// TwinCAT 3 PLC project HPT_PLC
// Title: Hardpoint Test Stand
// Company: GTMO
// Author: A. Everman, T. Ranka
// ProjectVersion: 1.4.5
// ProgramVersion: 3.1.4024.12
// libraries:
//   CmpBitmapPool, * (System)
//   Tc2_ControllerToolbox, * (Beckhoff Automation GmbH)
//   Tc2_EtherCAT, * (Beckhoff Automation GmbH)
//   Tc2_SerialCom, * (Beckhoff Automation GmbH)
//   Tc2_Standard, * (Beckhoff Automation GmbH)
//   Tc2_System, * (Beckhoff Automation GmbH)
//   Tc2_Utilities, * (Beckhoff Automation GmbH)
//   Tc3_Module, * (Beckhoff Automation GmbH)
// project tree:
//   DUTs/ ImagePool.TcIPO (not stored)
//   / Fast.TcTTO, GlobalTextList.TcGTLO, PlcTask.TcTTO, Visualization Manager.TcVMO (not stored)
//   GVLs/ GVL_TS.TcGVL
//   POUs/ FB_AirConv.TcPOU, Background.TcPOU, BackgroundEL.TcPOU, FB_BinToVer.TcPOU, FB_ClearFault.TcPOU, FB_CountConv.TcPOU, FB_PLCTime.TcPOU, FB_PyListener.TcPOU, FB_PyListenerStiffness.TcPOU, FB_PyPosRep.TcPOU, FB_ReadAlias.TcPOU, FB_ReadNcyl.TcPOU, FB_ReadSig.TcPOU, FB_readtextfile.TcPOU, FB_SAstiffness.TcPOU, FB_SaveData.TcPOU, FB_SerialCom.TcPOU, FB_HeidConv.TcPOU, FB_TriForce.TcPOU, FB_WriteHPTSettings.TcPOU, FB_WritePWM.TcPOU, FB_WriteSDO.TcPOU, MAIN.TcPOU, FB_MtrCtrl.TcPOU, FB_PLoop.TcPOU, FB_ROMTest.TcPOU, FB_SineSweep.TcPOU
// real-time tasks:
//   TASK PlcTask: cycle T#1ms, priority 6, ADS port 350
//   TASK Fast: cycle T#1ms, priority 4, ADS port 351
// motion (NC):
//   TASK NC-Task 1 SAF: cycle T#2ms, priority 8, ADS port 501
//   TASK NC-Task 1 SVB: cycle T#10ms, priority 12, ADS port 511
//   AXIS Axis 1 (id 1)
//     OtherSettings: AllowMotionCmdToSlave=true
//     encoder EncType=19
//       EncPara: MaxCount=#xffffffff
//     drive DrvType=16
//       DrvPara: MaxCount=#xffffffff
//         Analog: TorqueSetpointScale=10, ScaleFactorActTorque=0.1
//         TimeComp: TaskDelayCycles=1
//     controller CtrType=1
//       CtrPara: PriorControlFactor=1
//         Observer: BandWidth=20
// I/O:
//   DEVICE Device 1 (EtherCAT), AmsNetId 10.10.160.129.2.1
//     Term 2 (EK1100) [EK1100 EtherCAT Coupler (2A E-Bus)]
//       Term 13 (EL6070-0033) [EL6070-0033 1Ch. Licence key terminal, individual licences]
//       Term 14 (EL4102) [EL4102 2Ch. Ana. Output  0-10V, 16bit]
//       Term 16 (EL3002) [EL3002 2Ch. Ana. Input +/-10V]
//       Term 18 (EL3052) [EL3052 2Ch. Ana. Input 4-20mA]
//       Term 19 (EL5101) [EL5101 1Ch. Inc. Encoder 5V]
//       Term 29 (EL9011) [EL9011 End Terminal]
//     Drive 20 (BEL) [BEL]
//       modules: Module 1 (Cyclic velocity Mode)
//     Term 21 (EK1100) [EK1100 EtherCAT Coupler (2A E-Bus)]
//       Term 22 (EL5042) [EL5042 2Ch. BiSS-C Encoder]
//       Term 23 (EL3312) [EL3312 2Ch. Ana. Input Thermocouple (TC)]
//       Term 24 (EL9505) [EL9505 Power supply terminal 5V]
//       Term 26 (EL3356-0010) [EL3356-0010 1Ch. Ana. Input Resistor Bridge Terminal, 24bit, High Precision]
//       Term 30 (EL9011) [EL9011 End Terminal]
//     Box 17 (m1sa) [m1sa]
// variable links:
//   HPT_PLC/HPT_PLC Instance <-> Device 1 (EtherCAT)/Box 17 (m1sa)
//     PlcTask Inputs/MAIN.err_cal <-> Status process data mapping/MAIN.err_cal
//     PlcTask Inputs/MAIN.err_dongle <-> Status process data mapping/MAIN.err_dongle
//     PlcTask Inputs/MAIN.err_f_minmax <-> Status process data mapping/MAIN.err_f_minmax
//     PlcTask Inputs/MAIN.err_f_step <-> Status process data mapping/MAIN.err_f_step
//     PlcTask Inputs/MAIN.err_locid <-> Status process data mapping/MAIN.err_locid
//     PlcTask Inputs/MAIN.err_mhb <-> Status process data mapping/MAIN.err_mhb
//     PlcTask Inputs/MAIN.err_soc <-> Status process data mapping/MAIN.err_soc
//     PlcTask Inputs/MAIN.pwm1 <-> Status process data mapping/MAIN.pwm1
//     PlcTask Inputs/MAIN.rb_x <-> Status process data mapping/MAIN.rb_x
//     PlcTask Inputs/MAIN.spr_x <-> Status process data mapping/MAIN.spr_x
//     PlcTask Outputs/MAIN.close_loop <-> Control process data mapping/MAIN.close_loop
//     PlcTask Outputs/MAIN.enable <-> Control process data mapping/MAIN.enable
//     PlcTask Outputs/MAIN.msthb <-> Control process data mapping/MAIN.msthb
//     PlcTask Outputs/MAIN.sp_x <-> Control process data mapping/MAIN.sp_x
//   HPT_PLC/HPT_PLC Instance <-> Device 1 (EtherCAT)/Drive 20 (BEL)
//     PlcTask Inputs/GVL_TS.DIO_status <-> Transmit PDO 4/GVL_TS.DIO_status
//     PlcTask Inputs/GVL_TS.EncoderFault <-> Transmit PDO 3/GVL_TS.EncoderFault
//     PlcTask Inputs/GVL_TS.Sticky <-> Transmit PDO 4/GVL_TS.Sticky
//     PlcTask Inputs/GVL_TS.cmdVel <-> Transmit PDO 1/GVL_TS.cmdVel
//     PlcTask Inputs/GVL_TS.mtrCurrent <-> Transmit PDO 3/GVL_TS.mtrCurrent
//     PlcTask Inputs/GVL_TS.mtr_pos <-> Transmit PDO 2/GVL_TS.mtr_pos
//     PlcTask Inputs/GVL_TS.mtr_tor <-> Module 1 (Cyclic velocity Mode)/Cyclic velocity Inputs/GVL_TS.mtr_tor
//     PlcTask Inputs/GVL_TS.mtrl_vel <-> Module 1 (Cyclic velocity Mode)/Cyclic velocity Inputs/GVL_TS.mtrl_vel
//     PlcTask Inputs/GVL_TS.status_word <-> Module 1 (Cyclic velocity Mode)/Cyclic velocity Inputs/GVL_TS.status_word
//     PlcTask Outputs/GVL_TS.ClearLatched2181 <-> Receive PDO 4/GVL_TS.ClearLatched2181
//     PlcTask Outputs/GVL_TS.ClearLatched2183 <-> Receive PDO 4/GVL_TS.ClearLatched2183
//     PlcTask Outputs/GVL_TS.StopAbort <-> Receive PDO 3/GVL_TS.StopAbort
//     PlcTask Outputs/GVL_TS.TransitionFromQS <-> Receive PDO 3/GVL_TS.TransitionFromQS
//     PlcTask Outputs/GVL_TS.control_word <-> Module 1 (Cyclic velocity Mode)/Cyclic velocity Outputs/GVL_TS.control_word
//     PlcTask Outputs/GVL_TS.target_vel <-> Module 1 (Cyclic velocity Mode)/Cyclic velocity Outputs/GVL_TS.target_vel
//     PlcTask Outputs/MAIN.FaultMask <-> Receive PDO 3/MAIN.FaultMask
//   HPT_PLC/HPT_PLC Instance <-> Device 1 (EtherCAT)/Term 2 (EK1100)/Term 14 (EL4102)
//     PlcTask Outputs/GVL_TS.AirOut1 <-> Channel 1/GVL_TS.AirOut1
//     PlcTask Outputs/GVL_TS.AirOut2 <-> Channel 2/GVL_TS.AirOut2
//   HPT_PLC/HPT_PLC Instance <-> Device 1 (EtherCAT)/Term 2 (EK1100)/Term 16 (EL3002)
//     PlcTask Inputs/GVL_TS.LazrStrength <-> AI Standard Channel 1/GVL_TS.LazrStrength
//   HPT_PLC/HPT_PLC Instance <-> Device 1 (EtherCAT)/Term 2 (EK1100)/Term 18 (EL3052)
//     PlcTask Inputs/GVL_TS.FlowIn <-> AI Standard Channel 2/GVL_TS.FlowIn
//     PlcTask Inputs/GVL_TS.PressureIn <-> AI Standard Channel 1/GVL_TS.PressureIn
//   HPT_PLC/HPT_PLC Instance <-> Device 1 (EtherCAT)/Term 21 (EK1100)/Term 22 (EL5042)
//     PlcTask Inputs/GVL_TS.ActEncCount <-> FB Inputs Channel 1/GVL_TS.ActEncCount
//     PlcTask Inputs/GVL_TS.MirEncCount <-> FB Inputs Channel 2/GVL_TS.MirEncCount
//   HPT_PLC/HPT_PLC Instance <-> Device 1 (EtherCAT)/Term 21 (EK1100)/Term 23 (EL3312)
//     PlcTask Inputs/GVL_TS.EncTapeTemp <-> TC Inputs Channel 1/GVL_TS.EncTapeTemp
//     PlcTask Inputs/GVL_TS.MotorTemp <-> TC Inputs Channel 2/GVL_TS.MotorTemp
//   HPT_PLC/HPT_PLC Instance <-> Device 1 (EtherCAT)/Term 21 (EK1100)/Term 26 (EL3356-0010)
//     PlcTask Inputs/GVL_TS.LC_InR <-> RMB Value (Real)/GVL_TS.LC_InR

CONFIGURATION HPT_PLC
    RESOURCE PLC ON TwinCAT3
        TASK Fast(INTERVAL := T#1ms, PRIORITY := 4);
        TASK PlcTask(INTERVAL := T#1ms, PRIORITY := 6);
        PROGRAM Background WITH Fast : Background;
        PROGRAM MAIN WITH PlcTask : MAIN;
    END_RESOURCE
END_CONFIGURATION

// ---- GVLs/GVL_TS.TcGVL
VAR_GLOBAL CONSTANT
	max_rows : UDINT := 10001;
END_VAR

{attribute 'qualified_only'}
VAR_GLOBAL

// Variables for EL4102 0-10V Module for Air Control
AirOut1 AT %Q*			: INT;
AirOut2 AT %Q*			: INT;

// Variables for EL5101 RS422 Incremental Encoder Interface
RSCount AT %I* 			: DINT;
CountReset AT %Q* 		: DINT; // Count reset variable, set to zero for tareing of laser interferometer 
CountResetEn AT %Q* 	: BOOL; // Enable flag for counter reset
LaserUnder AT %I* 		: BOOL; // Underflow flag for debugging
LaserOver AT %I* 		: BOOL; // Overflow flag for debugging

// Variables for HPT eBox EL5042 BiSS-C Encoder Interface
ActEncCount AT %I* 		: ULINT;
MirEncCount AT %I* 		: ULINT;

// Motor variables
mtr_tor AT %I* 			: INT;
StopAbort AT %Q* 		: INT;
TransitionFromQS AT %Q* : INT;
mtrCurrent AT %I* 		: INT;
control_word AT %Q* 	: UINT;
status_word AT %I* 		: UINT;
target_vel AT %Q* 		: DINT :=0; (*0.1cnts/s*)
mtrl_vel AT %I* 		: DINT; (*0.1cnts/sec*)
mtr_pos AT %I* 			: DINT; (*counts*)
velLoopErr AT %I*		: DINT;
cmdVel AT %I*			: DINT;
ClearLatched2181 AT %Q* : UDINT;
ClearLatched2183 AT %Q* : UDINT;
Sticky AT %I* 			: UDINT;
EncoderFault AT %I* 	: UDINT;
DIO_status AT %I* 		: UDINT;	(*limit switch status*)
bLim_pos 				: BOOL := FALSE;
bLim_neg 				: BOOL := FALSE;
bEnableState 			: BOOL;
bReset 					: BOOL;
bEnable 				: BOOL;
sJog 					: STRING;

// Load cell input variable
LC_InR AT %I* 			: REAL;
LC_Tara AT %Q*			: BYTE;

// Thermocouple Variables
EncTapeTemp AT %I* 		: INT;
MotorTemp AT %I* 		: INT;

// Limit switch triggered status variables
bPos 					: BOOL;
bNeg 					: BOOL;
Pdiff 					: LREAL;

// EL3002 Interferometer Laser Strength Indicator Variable
LazrStrength AT %I* 	: INT;

// EL3052 4...20mA analog input variables for pressure/flow sensors
PressureIn AT %I* 		: INT;
FlowIn AT %I* 			: INT;

// Buffer variable for RS-232 COM port
RxBufferEL				: ComBuffer;	(* Receive data buffer; used with all receive function blocks *)
TxBufferEL				: ComBuffer;	(* Transmit data buffer; used with all receive function blocks *)

(* DEBUG VARIABLES *)
//bTEST1 				: BOOL := FALSE;
//bTEST2 				: BOOL := FALSE;
//wTest 				: WORD;
//sTest 				: STRING;

END_VAR

// ---- POUs/Background.TcPOU
PROGRAM Background
VAR
END_VAR

(*
The SerialLineControl function block is supposed to be called in every PLC cycle.
It communicates with the serial line hardware device and transmits or receives data.
The SerialLineControl can be called in the standard task (e.g.for PcCOM port usage) 
or in a separate fast task (e.g.for terminal usage) as well.
A fast separate task will be necessary at high baud rates or with KL6001 terminals 
which have a small process image (3 or 5 data bytes only)
*)

(* background communication with the EL6001 terminal *)
BackgroundEL();

END_PROGRAM

// ---- POUs/BackgroundEL.TcPOU
PROGRAM BackgroundEL
VAR
	(* background communication with the EL6001 terminal *)
	fbEL6001Ctrl		: SerialLineControl;
	bEL6001CtrlError	: BOOL;
	eEL6001CtrlErrorID	: ComError_t;
	(* 	I/O variables for a EL6001 terminal*)
	stIn_EL6001 AT %I*	: EL6inData22B;	(* linked to the EL6001 in the TwinCAT System Manager *)
	stOut_EL6001 AT %Q*	: EL6outData22B;(* linked to the EL6001 in the TwinCAT System Manager *)
END_VAR

(*
The SerialLineControl function block is supposed to be called in every PLC cycle.
It communicates with the serial line hardware device and transmits or receives data.
The SerialLineControl can be called in the standard task (e.g.for PcCOM port usage) 
or in a separate fast task (e.g.for terminal usage) as well.
A fast separate task will be necessary at high baud rates or with KL6001 terminals 
which have a small process image (3 or 5 data bytes only)
*)

(* background communication with the EL6001 terminal *)
fbEL6001Ctrl(
	Mode:= SERIALLINEMODE_EL6_22B, 
	pComIn:= ADR(stIn_EL6001), 
	pComOut:= ADR(stOut_EL6001), 
	SizeComIn:= SIZEOF(stIn_EL6001), 
	Error=> , 
	ErrorID=> , 
	TxBuffer:= GVL_TS.TxBufferEL, 
	RxBuffer:= GVL_TS.RxBufferEL );
IF fbEL6001Ctrl.Error THEN
	bEL6001CtrlError := TRUE;
	eEL6001CtrlErrorID := fbEL6001Ctrl.ErrorID;
END_IF

END_PROGRAM

// ---- POUs/MAIN.TcPOU
PROGRAM MAIN
VAR

// Function instants
	fbSAstiffness		: FB_SAstiffness;
	fbWriteSettings		: FB_WriteHPTSettings;
	fbROM 				: FB_ROMTest;
	fbSWEEP 			: FB_SineSweep;
	fbSTIFF 			: FB_TriForce;
	fbBWY				: FB_TriForce;
	fbPLOOP 			: FB_PLoop;
	fbToString 			: FB_FormatString;
	fbB2V 				: FB_BinToVer;
	fbEL6001 			: FB_SerialCom;
	fbHeidCon 			: FB_HeidConv;
	fbPyListen			: FB_PyListener;
	fbPyListenStiff		: FB_PyListenerStiffness;
	fbWriteSDO			: FB_WriteSDO;
	fbGetTime			: FB_PLCTime;
	fbPyPosRep			: FB_PyPosRep;
	
// Startup Variables
	FaultMask AT %Q* 	: UDINT := 2#00000000;
	
// HMI Variables
	txtLazer 			: STRING;
	txtActEncVal 		: STRING;
	txtMirEncVal 		: STRING;
	txtRPM 				: STRING;
	txtTorque 			: STRING;
	BinStatus 			: STRING;
	txtActROM 			: STRING;
	txtMirROM 			: STRING;
	txtEngActEnc 		: STRING; 
	txtEngMirEnc 		: STRING;
	txtActMid 			: STRING;
	txtMirMid 			: STRING;
	txtLC 				: STRING;
	txtPdiff 			: STRING;
	txtBWYPress 		: STRING;
	txtFlow 			: STRING;
	txtMtrTemp			: STRING;
	txtEncTemp			: STRING;
	txtMtrCurrent		: STRING;
	sHeidOut 			: STRING;
	HeidA 				: STRING;
	HeidB 				: STRING;
	HeidC 				: STRING;
	HeidD 				: STRING;
	sSetpoint 			: STRING;
	sSelHPT				: STRING;
	sTime				: STRING;
	sp_force 			: STRING;
	engActEnc 			: LREAL; // Converted engineering units
	engMirEnc 			: LREAL; // Converted engineering units
	mtrRPM 				: LREAL;
	BWYPressPSI			: REAL;
	FlowRate 			: REAL;
	mtrTorq 			: REAL;
	mtrCurrent			: REAL;
	LazrMeter 			: REAL;
	AIR_CTR 			: REAL;
	ROM_Act 			: REAL;
	ROM_mirr			: REAL;
	HeidANum 			: REAL;
	HeidBNum 			: REAL;
	HeidCNum 			: REAL;
	HeidDNum 			: REAL;
	COARSE_VAL 			: REAL; // Variables for converted interferometer converted counts to length
	FINE_VAL 			: REAL;
	MtrTemp				: REAL;
	EncTemp				: REAL;
	TestCycles			: INT;
	atto1 				: REAL;
	atto2 				: REAL;
	atto3 				: REAL;
	atto4 				: REAL;
	atto5 				: REAL;
	atto6 				: REAL;
	atto1uM 			: REAL;
	atto2uM 			: REAL;
	atto3uM 			: REAL;
	atto4uM 			: REAL;
	atto5uM 			: REAL;
	atto6uM 			: REAL;
	satto1uM 			: STRING;
	satto2uM 			: STRING;
	satto3uM 			: STRING;
	satto4uM 			: STRING;
	satto5uM 			: STRING;
	satto6uM 			: STRING;
	ROM_ActMid 			: ULINT;
	ROM_MirrMid 		: ULINT;
	btnEnb 				: BOOL;
	btnEnbnum 			: BOOL := FALSE;
	btnReset 			: BOOL := FALSE;
	btnTareLC			: BOOL := FALSE;
	btnPyPosRep			: BOOL := FALSE;
	btnClrSAerrors		: BOOL := FALSE; 
	tglSine 			: BOOL := FALSE;
	tglROM 				: BOOL := FALSE;
	tglStiffness 		: BOOL := FALSE;
	tglSAstiffness		: BOOL := FALSE;
	tglBWY				: BOOL := FALSE;
	tglPLoop 			: BOOL := FALSE;
	tglPyTest			: BOOL := FALSE;
	JogPos 				: BOOL := FALSE;
	JogNeg 				: BOOL := FALSE;
	PyLoad				: BOOL;
	PyLoadBusy			: BOOL := FALSE;
	PyEnable			: BOOL := TRUE;
	MtrErrArr 			: ARRAY[0..15] OF BOOL;
	
(* DEBUG VARIABLES *)
	//test 				: BOOL := FALSE;
	//int1 				: INT;
	//real2 			: REAL;
	//real3 			: REAL;
	
// SA Related Variables for Stiffness Fixture
	// actions
	actions : (idle, clear_all, enable_all, disable_all,read_ncyl,read_alias,read_gains,write_gains,read_file,send_waveform_cmd, send_waveform_cmd_debug, send_waveform_pwm);
	sp_x AT %Q* : REAL;
	sp_y AT %Q* : REAL;
	sp_z AT %Q* : REAL;
	
	f_num : INT := 1; // file number
	signal_scale : REAL := 1;
	signal_offset : REAL :=0;
	signal_axis : INT :=1;

	//VARIABLES FOR SENSOR OUTPUTS TO BE DISPLAYED IN UNITS OF MEASUREMENT
	spr_x AT %I* : REAL;
	spr_y AT %I* : REAL;
	spr_z AT %I* : REAL;
	rb_x AT %I* : REAL;
	txtRB_X 	: STRING;
	rb_y AT %I* : REAL;
	rb_z AT %I* : REAL;
	pwm1 AT %I* : REAL;
	pwm2 AT %I* : REAL;
	pwm3 AT %I* : REAL;
	cyl_sum : REAL;
	cmd_sum : REAL;
	
	//CONSTANTS FOR ADC GAIN COEFFICIENTS
	//ADC1: CH1 and CH2 PRESSURE, CH3 FLOW, CH4 NOT CONNECTED
	//ADC2: ALL CHANNELS PRESSURE
	GAIN_PRESSURE : REAL := 2.2;
	GAIN_FLOW : REAL := 2.2;//80;
	
	// ***********************************************************
	
	sa_addr : UINT := 1013;	
	clearfault : FB_ClearFault;
	readncyl : FB_ReadNcyl;
	readalias : FB_ReadAlias;
	readfile : FB_readtextfile;
	
	max_rows : UDINT := 10001;
	sfile : T_MaxString ;
	waveform_pwm : FB_WritePWM;
	state : INT := 2;
	step : DWORD :=0;
	bError : BOOL;
	t_index : UINT :=1;
	alias : UDINT;
	ncyl: UINT;
	signal : ARRAY[1.. GVL_TS.max_rows] OF REAL;
	
	fol_err : REAL;
	db : REAL := 14.0;
	dbi : REAL := 0;
	pwm : REAL := 0.0;
	value : REAL := 0.0;
	
	sdo_address: UINT;
	subIndex: BYTE;
	sNetId_local : T_AmsNetId := '10.134.198.192.2.1';	// Address of this computer 
	//sNetId_local : T_AmsNetId := '10.10.16.19.2.1';	// Address of this computer
	
// heartbeat
	msthb AT %Q* : UDINT;
	enable AT %Q* : BOOL;
	close_loop AT %Q* : BOOL;
	
	err_mhb AT %I* : BOOL;
	err_f_minmax AT %I* : BOOL;
	err_f_step AT %I* : BOOL;
	err_cal AT %I* : BOOL;
	err_dongle AT %I* : BOOL;
	err_locid AT %I* : BOOL;
	err_soc AT %I* : BOOL;
	err_ff AT %I* : BOOL;
	
	force : INT;

END_VAR

(*-----------------------------------------------------------------------------------------------------
 	Hardpoint Test Stand, GMTO
 	v2.2.0
	
	*CHANGE LOG*
	1.0.0
			- First "complete" release
				-HMI
					-Control and monitor all sensors and tests
				-Scope project
					-Monitor and record all availible sensors and ADS variables and export as CSV for analysis
				-Tests included:
					-Range of motion
					-Position loop
					-Stiffness test
						-Multiple force profiles availible
					-Sine sweep
						*NOT TESTED ON HARDWARE, WORKS IN SCOPE PROJECT ONLY*
					
	1.4.5: 
			- Refactoring started:
				Clean up variables by standardizing naming conventions (upper camel case, leading lowercase b, s, fb, etc. for special case variables) 
				Whitespaces in declarations
				Removing unused variables
				Change variable types to lower memory footprint
				Reorganize variables to group by type
				
	1.4.6
			- Thermocouple data added to HMI
				Settings made in EL3312 to read correctly:
					CoE 8000:01 = TRUE
						8000:07 = TRUE
						8000:08 = TRUE
						8000:12 = 31451
						8000:13 = -730
						8000:14 = 4820
						8010:01 = TRUE
						8010:07 = TRUE
						8010:08 = TRUE
						8010:12 = 31438
						8010:13 = -730
						8010:14 = 4820
			- Further refactoring
			- Divided MAIN into clearer sections for ease of reading
			- Removed redundant limit switch check
			- Changed some HMI readouts to 4 decimal places
			
	1.4.7
			- HMI Cleanup and fixes
			- NOTE ADDED: EL5042 changes to be made to enable correct operation
				CoE 8008:15 - 26
					8008:16 - 0
					8018:15 - 26
					8018:16 - 0
	
	1.4.8	
			-= VERSION SKIPPED =-
	
	1.4.9	
			- Added, then removed, auto-tare for interferometer and load cell on test starts 
			- Added Tare button to HMI; disabled for time being
	
	2.0.0	
			- Python "PyListener" code added to listen for TC3 variables over ADS and build .CSV
				- Also grabs AttoCube measurements to calculate stiffness
			- Added ability to tare load cell back into HMI
				- Uses new FB_WriteSDO POU to write to SDOs in order to accomplish this
			- Added seperate buttons for both stiffness and breakaway tests
			- Simplified underlying stiffness/breakaway test code into one, singular function
				- Able to define both slope and force as inputs to function
			- Partitioned off tests into distinct "types" on HMI
			- Removed "Sine Sweep" test button from HMI; did not remove underlying code
				- CME has the ability to run bandwith tests natively, will need to add back into stand eventually
			- Further refactoring done to clean up unused variables/functions
			
	2.1.0
			- Python "PyListener" launches on start of any test, and ends collection on test stop
			- Further refactoring
			- Converted PLC time code into POU to clean up MAIN
	2.2.0
			- Added ability to toggle PyListener on and off
				- Buttons added on HMI for this
			- Able to launch PyListener for arbitrary data collection
			- Added cycle counter for stiffness/breakaway tests and readout on HMI
			- HMI cleaned up for better readability
			- HMI size property fixed to always show full dashboard when undocked
				
				
	TO-DO:
			
			- Use new FB_WriteSDO to force write all required settings on startup
				- Needs ability to write different variable sizes/types to correct positions
			- Continue refactoring as needed
			- Write new POU force stiffness/breakaway tests that has a "ramp up/hold/ramp down/hold/repeat profile"
				with ability to fully customize ramp speeds, hold times, and total force applied during all phases of test run
			- Possibly write a fully automated, non-steady state position loop test (I.E. start at set point, move up XXXcts, 
				return to starting setpoint, move down XXXcts, return to setpoint; do for how ever many cycles, each cycle
				being YYY[s] long)
			- Test/Debug Sine Sweep test on actual hardware
			- ??? (add to as necessary)

(*-----------------------------------------------------------------------------------------------------*)
 	Austin Everman - Overall framework, HMI, integration of code for individual tests, PyListener (with
	Trupti Ranka - coding for individual tests, technical help
	William Schoenell - AttoCube Python connection code

              _______________
          ==c(___(o(______(_()
                  \=\
                   )=\
                  //|\\
                 //|| \\
                // ||  \\
               //  ||   \\
              //         \\
			  
-------------------------------------------------------------------------------------------------------*)
(*-----------------------------------------------------------------------------------------------------*)
//fbWriteSettings();
(*-----------------------------------------------------------------------------------------------------*)
(* CONVERSION SECTION OF THE HMI THAT DEALS WITH TAKING RAW DATA AND CONVERTING IT FOR *)
(* DISPLAY ON THE DASHBOARD 														   *)
(*-----------------------------------------------------------------------------------------------------*)
// Parse status word into boolean array for HMI
fbB2V(
	BinInput := GVL_TS.status_word, 
	MtrErrArr => MtrErrArr
);
(*-----------------------------------------------------------------------------------------------------*)
// Convert interferometer signal strength voltage output to scaled 0-100% output for HMI
LazrMeter := (INT_TO_REAL(GVL_TS.LazrStrength)/32767) * 1000;
(*-----------------------------------------------------------------------------------------------------*)
// Call function to convert interferometer counts to mm
FB_CountConv(
	GVL_TS.RsCount, 
	MEASC_OUT => COARSE_VAL, // Return from function for conversion for coarse resolution laser intererometric measurements; Currently in use
	MEASF_OUT => FINE_VAL    // Not in use, but conversion made for fine resolution in event of use; setting is made on RLU dip switch on front of unit
);
(*-----------------------------------------------------------------------------------------------------*)
// Convert coarse interferometer value to string, limit to 6 decimal places for HMI, include 'traveling' engineering unit
fbToString(
	sFormat := '%.6f', 
	arg1 := F_REAL(COARSE_VAL), 
	sOut => txtLazer
);
txtLazer := CONCAT(txtLazer, ' mm');
(*-----------------------------------------------------------------------------------------------------*)
// Convert encoder values to string for HMI
txtActEncVal := TO_STRING(GVL_TS.ActEncCount);
txtMirEncVal := TO_STRING(GVL_TS.MirEncCount);
(*-----------------------------------------------------------------------------------------------------*)
// Convert actuator and mirror encoder counts to engineering units (mm) and display only 4 decimal places
engActEnc := GVL_TS.ActEncCount * 5E-6;
fbToString(
	sFormat := '%.5f', 
	arg1 := F_LREAL(engActEnc), 
	sOut => txtEngActEnc
);
txtEngActEnc := CONCAT(txtEngActEnc, ' mm');
engMirEnc := GVL_TS.MirEncCount * 5E-6;
fbToString(
	sFormat := '%.5f', 
	arg1 := F_LREAL(engMirEnc), 
	sOut => txtEngMirEnc
);
txtEngMirEnc := CONCAT(txtEngMirEnc, ' mm');
txtActMid := TO_STRING(ROM_ActMid);
txtMirMid := TO_STRING(ROM_MirrMid);

// Limit encoder range displayed on HMI to 4 decimal places
fbToString(
	sFormat := '%.4f', 
	arg1 := F_REAL(ROM_Act), 
	sOut => txtActROM
);
txtActROM := CONCAT(txtActROM, ' mm');
fbToString(
	sFormat := '%.4f', 
	arg1 := F_REAL(ROM_mirr), 
	sOut => txtMirROM
);
txtMirROM := CONCAT(txtMirROM, ' mm');
(*-----------------------------------------------------------------------------------------------------*)
// Read out reported velocity from motor and convert using scaling factor into string; tack on RPM string 
// at the end to make it all fancy-like
// Scale factor = (1 revolution/2^17 counts)(0.1 counts/second)(60 seconds/minute)
mtrRPM := TO_LREAL(GVL_TS.mtrl_vel) * 4.578E-5;
fbToString(
	sFormat := '%.3f', 
	arg1 := F_LREAL(mtrRPM), 
	sOut => txtRPM
);
txtRPM := CONCAT(txtRPM, ' RPM');
(*-----------------------------------------------------------------------------------------------------*)
// Read out torque value from motor, convert to engineering units, and tack on travelling unit
// for HMI display like previous conversions
mtrTorq := GVL_TS.mtr_tor; // NEEDS CONVERSION FACTOR!!!!!!
fbToString(
	sFormat := '%.3f', 
	arg1 := F_REAL(mtrTorq), 
	sOut => txtTorque
);
txtTorque := CONCAT(txtTorque, ' Nm');
(*-----------------------------------------------------------------------------------------------------*)
// Read out torque value from motor, convert to engineering units, and tack on travelling unit
// for HMI display like previous conversions
mtrCurrent := (TO_REAL(GVL_TS.mtrCurrent)) / 100; // NEEDS CONVERSION FACTOR!!!!!!
fbToString(
	sFormat := '%.3f', 
	arg1 := F_REAL(mtrCurrent), 
	sOut => txtMtrCurrent
);
txtMtrCurrent := CONCAT(txtMtrCurrent, ' A');
(*-----------------------------------------------------------------------------------------------------*)
// Limit loadcell display on HMI to 4 decimal places and tack on traveling 'N' engineering unit at end
fbToString(
	sFormat := '%.4f', 
	arg1 := F_REAL(GVL_TS.LC_InR), 
	sOut => txtLC
);
txtLC := CONCAT(txtLC, ' N');
(*-----------------------------------------------------------------------------------------------------*)
// Convert the difference in PID setpoint and actuator count into string for display on HMI
fbToString(
	sFormat := '%.0f', 
	arg1 := F_LREAL(GVL_TS.Pdiff), 
	sOut => txtPdiff
);
txtPdiff := CONCAT(txtPdiff, ' Cts');
(*-----------------------------------------------------------------------------------------------------*)
// Convert input pressure from Bar to PSI then into string for display on HMI
BWYPressPSI := (10 * (TO_REAL(GVL_TS.PressureIn) / 32767)) * 14.504;
fbToString(
	sFormat := '%.3f', 
	arg1 := F_REAL(BWYPressPSI), 
	sOut => txtBWYPress
);
txtBWYPress := CONCAT(txtBWYPress, ' PSI');
(*-----------------------------------------------------------------------------------------------------*)
// Convert flow rate into string for display on HMI
FlowRate := 20 * (TO_REAL(GVL_TS.FlowIn) / 32767);
fbToString(
	sFormat := '%.3f', 
	arg1 := F_REAL(FlowRate), 
	sOut => txtFlow
);
txtFlow := CONCAT(txtFlow, ' SLPM');
(*-----------------------------------------------------------------------------------------------------*)
// Convert thermocouple readings for display on HMI
MtrTemp := TO_REAL(GVL_TS.MotorTemp) / 10;
EncTemp := TO_REAL(GVL_TS.EncTapeTemp) / 10;

fbToString(
	sFormat := '%.1f', 
	arg1 := F_REAL(MtrTemp), 
	sOut => txtMtrTemp
);
txtMtrTemp := CONCAT(txtMtrTemp, ' C');

fbToString(
	sFormat := '%.1f', 
	arg1 := F_REAL(EncTemp), 
	sOut => txtEncTemp
);
txtEncTemp := CONCAT(txtEncTemp, ' C');
(*-----------------------------------------------------------------------------------------------------*)
(*-----------------------------------------------------------------------------------------------------*)
(*-----------------------------------------------------------------------------------------------------*)
(*									   *)
(* TEST AND CONTROL SECTION OF THE HMI *)
(*									   *)
(*-----------------------------------------------------------------------------------------------------*)
(*-----------------------------------------------------------------------------------------------------*)
(*-----------------------------------------------------------------------------------------------------*)
// Call function to convert slider position in HMI to EL4102 0-10V signal
FB_AirConv(AIR_CTR);
(*-----------------------------------------------------------------------------------------------------*)
// Enable the motor and set enable flag for the rest of the program
FB_MtrCtrl(
	bBtnEnb => btnEnb
);
(*-----------------------------------------------------------------------------------------------------*)
// If no tests running, set motor enable flag to flase, and run motor control routine to disable the motor
IF tglSine = FALSE AND tglROM = FALSE THEN
	FB_MtrCtrl();
END_IF
(*-----------------------------------------------------------------------------------------------------*)
// If HMI "Start Sine Sweep" button pressed, set enable motor flag, run motor control routine, and run sine sweep test
IF tglSine = TRUE THEN
	FB_MtrCtrl();
	fbSWEEP();	
END_IF
(*-----------------------------------------------------------------------------------------------------*)
// If HMI "Start Range of Motion Test" button pressed, set enable motor flag, run motor control routine, and run range of motion test
IF tglROM = TRUE THEN
	FB_MtrCtrl();
	fbROM(
		ROM_Act => ROM_Act, 
		ROM_mirr => ROM_mirr, 
		ROM_ActMid => ROM_ActMid, 
		ROM_MirrMid => ROM_MirrMid 
		);
ELSE
	GVL_TS.target_vel := 0;
	FB_MtrCtrl();
END_IF
(*-----------------------------------------------------------------------------------------------------*)
// If HMI "Reset Motor" button pressed, disable motor, enable motor reset flag, and run motor control routine to pass commands
IF btnReset = TRUE THEN
	GVL_TS.bReset := TRUE;
	FB_MtrCtrl();
END_IF
(*-----------------------------------------------------------------------------------------------------*)
// If HMI "Enable Motor" button pressed, set enable motor flag and run motor control routine
IF btnEnb = TRUE THEN
	FB_MtrCtrl();
END_IF
(*-----------------------------------------------------------------------------------------------------*)
// If either "Jog Position" button pressed, activate motor control with appropriate target velocity
IF JogPos = TRUE THEN
	FB_MtrCtrl();
	GVL_TS.target_vel := TO_DINT(STRING_TO_WORD(GVL_TS.sJog)/(4.578E-5));
END_IF

IF JogNeg = TRUE THEN
	FB_MtrCtrl();
	GVL_TS.target_vel := TO_DINT(STRING_TO_WORD(GVL_TS.sJog)/(-4.578E-5));
END_IF
(*-----------------------------------------------------------------------------------------------------*)
// Start Python data collection if any test is ran
IF (tglSAStiffness = TRUE OR tglStiffness = TRUE OR tglBWY = TRUE OR tglROM = TRUE OR tglSine = TRUE OR tglPLoop = TRUE OR tglPyTest = TRUE) AND PyEnable = TRUE THEN
	
	IF (tglStiffness = TRUE OR tglBWY = TRUE OR tglROM = TRUE OR tglSine = TRUE OR tglPLoop = TRUE) THEN
		fbPyListen(bExecute := TRUE);
	END_IF
	
	IF (tglSAStiffness = TRUE OR tglPyTest = TRUE) THEN
		fbPyListenStiff(bExecute := TRUE);
		PyLoadBusy := TRUE;
	END_IF
	PyLoadBusy := TRUE;
ELSE
	fbPyListen(
		Initialized := FALSE,
		bExecute := FALSE,
		Init_State := 0
	);
	fbPyListenStiff(
		Initialized := FALSE,
		bExecute := FALSE,
		Init_State := 0
	);
	PyLoadBusy := FALSE;
END_IF
(*-----------------------------------------------------------------------------------------------------*)

// If HMI "Start Stiffness Test" button pressed, disable motor enable flag, run motor control routine
// and start stiffness test
IF tglStiffness = TRUE THEN
	FB_MtrCtrl();
	fbSTIFF(
		Slope := 10000,
		Force := 7500, //Original force for 450N
		CyclesOut => TestCycles,
	);
ELSE
	fbSTIFF.Cycles := 0;
	fbSTIFF.Counter := 0;
	fbSTIFF.Channel1Command := 0;
	fbSTIFF.Channel2Command := 0;
END_IF
(*-----------------------------------------------------------------------------------------------------*)
// If HMI "Start Stiffness Test" button pressed, disable motor enable flag, run motor control routine
// and start stiffness test
IF tglBWY = TRUE THEN
	FB_MtrCtrl();
	fbBWY(
		Slope := 10000,
		Force := 32767,
		CyclesOut => TestCycles
	);
ELSE
	fbBWY.Cycles := 0;
	fbBWY.Counter := 0;
	fbBWY.Channel1Command := 0;
	fbBWY.Channel2Command := 0;
END_IF
(*-----------------------------------------------------------------------------------------------------*)
// Start motor control, convert setpoint value from string into number, and start position loop test
IF tglPLoop = TRUE THEN
	FB_MtrCtrl();
	fbPLOOP(
		fSetPointValue := STRING_TO_REAL(sSetpoint)
	);
END_IF
(*-----------------------------------------------------------------------------------------------------*)
// If "Tare Load Cell" button pressed, write to appropriate SDO to perform taring operation 
IF btnTareLC = TRUE THEN
	fbWriteSDO(
		nSlaveAddr := 1012,
		nIndex := 16#FB00,
		nSubIndex := 16#01,
		bExecute := TRUE,
		nValueInt := 16#02
		);
END_IF
(*-----------------------------------------------------------------------------------------------------*)
// If no tests are running, ensures motor is disabled
IF tglSAstiffness = FALSE AND tglSine = FALSE AND tglROM = FALSE AND tglStiffness = FALSE AND JogPos = FALSE AND JogNeg = FALSE THEN
	FB_MtrCtrl();
END_IF
(*-----------------------------------------------------------------------------------------------------*)
// Send and receive commands over the Heidenhain RS-232 interface
fbEL6001(
	TxBuffer := GVL_TS.TxBufferEL, 
	RxBuffer := GVL_TS.RxBufferEL, 
	sHeidOut => sHeidOut
);
// Convert the massive single string sent over RS-232 into 4 smaller strings for display on the HMI
fbHeidCon(
	sHeidIn := sHeidOut, 
	s1 => HeidA, 
	s2 => HeidB, 
	s3 => HeidC, 
	s4 => HeidD
);
// Convert each string into a REAL formatted number for data processing
HeidANum := STRING_TO_REAL(HeidA);
HeidBNum := STRING_TO_REAL(HeidB);
HeidCNum := STRING_TO_REAL(HeidC);
HeidDNum := STRING_TO_REAL(HeidD);
(*-----------------------------------------------------------------------------------------------------*)
// Get PLC time
fbGetTime(
	sTime => sTime
	);
(*-----------------------------------------------------------------------------------------------------*)
IF btnPyPosRep = TRUE THEN
	fbPyPosRep(bExecute := TRUE);
	FB_MtrCtrl();
	fbPLOOP(
		fSetPointValue := STRING_TO_REAL(sSetpoint)
	);
	PyLoadBusy := TRUE;
ELSE
	fbPyPosRep(
		Initialized := FALSE,
		bExecute := FALSE,
		Init_State := 0
	);
	//PyLoadBusy := FALSE;
END_IF
(*-----------------------------------------------------------------------------------------------------*)
(* BEGIN DEBUGGING CODE *)

// Convert drive amp status word from decimal to binary for display on HMI and easier debugging of problems
//ToString(sFormat := '%.16b', arg1 := F_UINT(GVL_TS.status_word), sOut => BinStatus);

// Tack on binary prefix notation, because I'm OCD like that ¯\_(ツ)_/¯
//BinStatus := CONCAT('0b', BinStatus);

(* END DEBUGGING CODE *)

(*-----------------------------------------------------------------------------------------------------*)
// SA RELATED CODE
(*-----------------------------------------------------------------------------------------------------*)

msthb := msthb + 1; // Increment masterheart count for SA
//fol_err := spr_x - rb_x;

CASE actions OF
	idle:
		state := 2;
		bError := 0;
		t_index := 1;
		sp_x := 0;
		sp_y := 0;
		sp_z := 0;
		
	enable_all :
		enable := TRUE;
		close_loop := TRUE;
		
	disable_all:
		enable := FALSE;
		close_loop := FALSE;
		
	clear_all:
	clearfault(bExecute := TRUE, 
		slv_addr := sa_addr, 
		state => state, 
		bError=> bError 
		);
		
	IF state = 0 THEN
		actions := idle;
	END_IF
		
	read_ncyl :
		readncyl(
			bExecute := TRUE, 
			slv_addr := sa_addr, 
			state => state, 
			bError=> bError, 
			value => ncyl 
			);
			
		IF state = 0 THEN
			actions := idle;
		END_IF
		
	read_alias :
		readalias(
			bExecute := TRUE, 
			slv_addr := sa_addr, 
			state => state, 
			bError=> bError, 
			value => alias 
			);
			
		IF state = 0 THEN
			actions := idle;
		END_IF
		
	read_file :
		CASE f_num OF
			1:
			sfile := 'C:\Users\gmto\Documents\TcXaeShell\signals\sine_0_1Hz_A1750.csv';
			max_rows := 10001;
			2:
			sfile := 'C:\Users\gmto\Documents\TcXaeShell\signals\sine_1Hz_A1750.csv';
			max_rows := 1001;
			3:
			sfile := 'C:\Users\gmto\Documents\TcXaeShell\signals\sine_3Hz_A1750.csv';
			max_rows := 334;
			4:
			sfile := 'C:\Users\gmto\Documents\TcXaeShell\signals\sine_5Hz_A1750.csv';
			max_rows := 201;
			5:
			sfile := 'C:\Users\gmto\Documents\TcXaeShell\signals\sine_10Hz_A1750.csv';
			max_rows := 101;
			6:
			sfile := 'C:\Users\gmto\Documents\TcXaeShell\signals\sinesweep_f1_50Hz_dt_1000Hz_amp15N_offset0.csv';
			max_rows := 11981;
			7:
			sfile := 'C:\Users\gmto\Documents\TcXaeShell\signals\sinesweep_f1_100Hz_dt_1000Hz_amp15N_offset0.csv';
			max_rows := 29995;
			8:
			sfile := 'C:\Users\gmto\Documents\TcXaeShell\signals\triangle.csv';
			max_rows := 10001;
			9:
			sfile := 'C:\Users\gmto\Documents\TcXaeShell\signals\sine_00_1Hz_A1750.csv';
			max_rows := 100001;
		END_CASE
		readfile(
			bRead := TRUE, 
			sFileName:=sfile, 
			output=>signal,
			step=>step
			);
			
		IF step = 0 THEN
			actions := idle;
		END_IF	
		
	send_waveform_cmd :
	CASE signal_axis OF
		1:
		sp_x := signal_scale * signal[t_index] + signal_offset;
		sp_y := 0;
		sp_z := 0;
		fol_err := spr_x - rb_x;
		2:
		sp_x := 0;
		sp_y := signal_scale * signal[t_index] + signal_offset;
		sp_z := 0;
		fol_err := spr_y - rb_y;
		3:
		sp_x := 0;
		sp_y := 0;
		sp_z := signal_scale * signal[t_index] + signal_offset;	
		fol_err := spr_z - rb_z;
	END_CASE
		t_index := t_index + 1;
		IF t_index > max_rows THEN
			t_index := 1;
		END_IF

	send_waveform_cmd_debug :
	CASE signal_axis OF
		1:
		sp_x := signal_scale*signal[t_index]+signal_offset;
		sp_y := 0;
		sp_z := 0;
		fol_err := spr_x - rb_x;
		2:
		sp_x := signal_scale * signal[t_index] + signal_offset;
		sp_y := signal_scale * signal[t_index] + signal_offset;
		sp_z := 0;
		fol_err := spr_y - rb_y;
		3:
		sp_x := signal_scale * signal[t_index] + signal_offset;
		sp_y := signal_scale * signal[t_index] + signal_offset;
		sp_z := signal_scale * signal[t_index] + signal_offset;	
		fol_err := spr_z - rb_z;
		4:
		sp_x := 0;
		sp_y := 0;
		sp_z := 0;
	END_CASE
	
		t_index := t_index+1;
		
		IF t_index>max_rows THEN
			t_index := 1;
		END_IF
	
	send_waveform_pwm:
		waveform_pwm(
			bExecute := TRUE, 
			slv_addr := sa_addr,
			value :=  signal[t_index], 
			state => state, 
			bError=> bError
			);
			
		t_index := t_index+1;
		
		IF t_index>max_rows THEN
			t_index := 1;
		END_IF
END_CASE

IF tglSAstiffness = FALSE THEN
	sp_x := STRING_TO_REAL(sp_force);
END_IF

IF tglSAstiffness = TRUE THEN
	fbSAstiffness(
		force => sp_x, 
		cyclesOut => TestCycles);
	sp_force := REAL_TO_STRING(sp_x);
	FB_MtrCtrl();
ELSE
	fbSAstiffness.cycles := 0;
	//fbSAstiffness.force := 0;
END_IF

IF btnClrSAerrors = TRUE THEN
	fbWriteSDO(
		nSlaveAddr := sa_addr,
		nSubIndex := 16#1,
		nIndex := 16#8006,
		nValueBool := 16#01,
		bExecute := TRUE);
END_IF

IF fbWriteSDO.bBusy = FALSE THEN
	fbWriteSDO.bExecute := FALSE;
END_IF

atto1uM := atto1 / 1000000; 
atto2uM := atto2 / 1000000; 
atto3uM := atto3 / 1000000; 
atto4uM := atto4 / 1000000; 
atto5uM := atto5 / 1000000; 
atto6uM := atto6 / 1000000;

fbToString(
	sFormat := '%.3f', 
	arg1 := F_REAL(atto1uM), 
	sOut => satto1uM
);
satto1uM := CONCAT(satto1uM, ' uM');

fbToString(
	sFormat := '%.3f', 
	arg1 := F_REAL(atto2uM), 
	sOut => satto2uM
);
satto2uM := CONCAT(satto2uM, ' uM'); 

fbToString(
	sFormat := '%.3f', 
	arg1 := F_REAL(atto3uM), 
	sOut => satto3uM
);
satto3uM := CONCAT(satto3uM, ' uM'); 

fbToString(
	sFormat := '%.3f', 
	arg1 := F_REAL(atto4uM), 
	sOut => satto4uM
);
satto4uM := CONCAT(satto4uM, ' uM'); 

fbToString(
	sFormat := '%.3f', 
	arg1 := F_REAL(atto5uM), 
	sOut => satto5uM
);
satto5uM := CONCAT(satto5uM, ' uM'); 

fbToString(
	sFormat := '%.3f', 
	arg1 := F_REAL(atto6uM), 
	sOut => satto6uM
);
satto6uM := CONCAT(satto6uM, ' uM'); 

fbToString(
	sFormat := '%.4f', 
	arg1 := F_REAL(rb_x), 
	sOut => txtRB_X
);
txtRB_X := CONCAT(txtRB_X, ' N');

END_PROGRAM

// ---- POUs/FB_SAstiffness.TcPOU
FUNCTION_BLOCK FB_SAstiffness
VAR_INPUT
	cycles : INT := 0;
END_VAR
VAR_OUTPUT
	cyclesOut : INT := 0;
	force : REAL := 0;
END_VAR
VAR
	counter : INT := 0;
	sign : REAL := 1;
END_VAR

counter := counter + 1;

IF counter = 50 THEN
	force := force + sign;
	counter := 0;
END_IF

IF force = 500 THEN
	sign := -1;
	cycles := cycles + 1;
END_IF

IF force = -500 THEN
	sign := 1;
	cycles := cycles + 1;
END_IF

cyclesOut := cycles;

END_FUNCTION_BLOCK

// ---- POUs/FB_WriteHPTSettings.TcPOU
FUNCTION_BLOCK FB_WriteHPTSettings
VAR_INPUT
END_VAR
VAR_OUTPUT
END_VAR
VAR
	WriteSetting	: FB_WriteSDO;
	Step			: INT := 1;
	Debug1			: BOOL;
	DebugSize2		: BYTE;
	err				: BOOL;
	errId			: UDINT;
END_VAR

CASE Step OF

1:
// Write Thermocouple Ch1 settings
WriteSetting(
	nSlaveAddr := 1011,
	nIndex := 16#8000,
	nSubIndex := 16#01,
	bExecute := TRUE,
	nValueBool := 16#01
);

Debug1 := TO_BOOL(WriteSetting.nValueBool);

IF WriteSetting.bBusy = FALSE THEN
	Step := Step +1;
END_IF

2:
WriteSetting(
	nSlaveAddr := 1011,
	nIndex := 16#8000,
	nSubIndex := 16#07,
	nValueBool := 16#01,
	bExecute := TRUE
);

IF WriteSetting.bBusy = FALSE THEN
	Step := Step +1;
END_IF

3:
WriteSetting(
	nSlaveAddr := 1011,
	nIndex := 16#8000,
	nSubIndex := 16#08,
	nValueBool := 16#01,
	bExecute := TRUE
);

IF WriteSetting.bBusy = FALSE THEN
	Step := Step +1;
END_IF

4:
WriteSetting(
	nSlaveAddr := 1011,
	nIndex := 16#8000,
	nSubIndex := 16#12,
	nValueDInt := 31451,
	bExecute := TRUE
);

IF WriteSetting.bBusy = FALSE THEN
	Step := Step +1;
END_IF

5:
WriteSetting(
	nSlaveAddr := 1011,
	nIndex := 16#8000,
	nSubIndex := 16#13,
	nValueInt := -730,
	bExecute := TRUE
);

IF WriteSetting.bBusy = FALSE THEN
	Step := Step +1;
END_IF

6:
WriteSetting(
	nSlaveAddr := 1011,
	nIndex := 16#8000,
	nSubIndex := 16#14,
	nValueInt := 4820,
	bExecute := TRUE
);

IF WriteSetting.bBusy = FALSE THEN
	Step := Step +1;
END_IF

7:
// Write Thermocouple Ch2 settings
WriteSetting(
	nSlaveAddr := 1011,
	nIndex := 16#8010,
	nSubIndex := 16#01,
	nValueBool := 16#01,
	bExecute := TRUE
);

IF WriteSetting.bBusy = FALSE THEN
	Step := Step +1;
END_IF

8:
WriteSetting(
	nSlaveAddr := 1011,
	nIndex := 16#8010,
	nSubIndex := 16#07,
	nValueBool := 16#01,
	bExecute := TRUE
);

IF WriteSetting.bBusy = FALSE THEN
	Step := Step +1;
END_IF

9:
WriteSetting(
	nSlaveAddr := 1011,
	nIndex := 16#8010,
	nSubIndex := 16#08,
	nValueBool := 16#01,
	bExecute := TRUE
);

IF WriteSetting.bBusy = FALSE THEN
	Step := Step +1;
END_IF

10:
WriteSetting(
	nSlaveAddr := 1011,
	nIndex := 16#8010,
	nSubIndex := 16#12,
	nValueDInt := 31451,
	bExecute := TRUE
);

IF WriteSetting.bBusy = FALSE THEN
	Step := Step +1;
END_IF

11:
WriteSetting(
	nSlaveAddr := 1011,
	nIndex := 16#8010,
	nSubIndex := 16#13,
	nValueInt := -730,
	bExecute := TRUE
);

IF WriteSetting.bBusy = FALSE THEN
	Step := Step +1;
END_IF

12:
WriteSetting(
	nSlaveAddr := 1011,
	nIndex := 16#8010,
	nSubIndex := 16#14,
	nValueInt := 4820,
	bExecute := TRUE,
	bError => err,
	nErrId => errid
);

(*
// Write EL5042 encoder settings to enable correct readout
WriteSetting(
	nSlaveAddr := 1010,
	nIndex := 16#8008,
	nSubIndex := 16#15,
	nValue := 26,
	bExecute := TRUE
);

WriteSetting(
	nSlaveAddr := 1010,
	nIndex := 16#8008,
	nSubIndex := 16#16,
	nValue := 0,
	bExecute := TRUE
);

WriteSetting(
	nSlaveAddr := 1010,
	nIndex := 16#8018,
	nSubIndex := 16#15,
	nValue := 26,
	bExecute := TRUE
);

WriteSetting(
	nSlaveAddr := 1010,
	nIndex := 16#8018,
	nSubIndex := 16#16,
	nValue := 0,
	bExecute := TRUE
);
*)
Step := 1;
END_CASE

END_FUNCTION_BLOCK

// ---- POUs/FB_WriteSDO.TcPOU
FUNCTION_BLOCK FB_WriteSDO
VAR_INPUT
        nSlaveAddr      : UINT; 
        nSubIndex       : BYTE; 
        nIndex          : WORD;
        pSrcBuf         : DWORD; 
        cbBufLen        : UDINT; 
        bExecute        : BOOL;
        tTimeout        : TIME := DEFAULT_ADS_TIMEOUT;
		nValueInt		: INT;
		nValueDInt		: UDINT;
		nValueBool		: BYTE;
END_VAR
VAR_OUTPUT
	    bBusy           : BOOL;
        bError          : BOOL;
        nErrId          : UDINT;
END_VAR
VAR
	fbSdoWriteInt      	: FB_EcCoESdoWrite;
	fbSdoWriteDInt      : FB_EcCoESdoWrite;
	fbSdoWriteBool      : FB_EcCoESdoWrite;
	sNetId          	: T_AmsNetId := '10.10.160.129.2.1'; (* NetId of EtherCAT Master *)

END_VAR

/////////////////////////////////////////////////////////
fbSdoWriteInt(
        sNetId          := sNetId,
        nSlaveAddr      := nSlaveAddr,
        nIndex          := nIndex,
        nSubIndex       := nSubIndex,
        pSrcBuf         := ADR(nValueInt),
        cbBufLen        := SIZEOF(nValueInt),
        bExecute        := bExecute
);

IF NOT fbSdoWriteInt.bBusy THEN
        bExecute := FALSE;
        IF NOT bError THEN 
                (* write successful *)
                bError := FALSE;
                nErrId := 0;
        ELSE 
                (* write failed *)
                bError := fbSdoWriteInt.bError;
                nErrId := fbSdoWriteInt.nErrId;
        END_IF

        fbSdoWriteInt(bExecute := FALSE);
END_IF
/////////////////////////////////////////////////////////
fbSdoWriteDInt(
        sNetId          := sNetId,
        nSlaveAddr      := nSlaveAddr,
        nIndex          := nIndex,
        nSubIndex       := nSubIndex,
        pSrcBuf         := ADR(nValueDInt),
        cbBufLen        := SIZEOF(nValueDInt),
        bExecute        := bExecute
);

IF NOT fbSdoWriteDInt.bBusy THEN
        bExecute := FALSE;
        IF NOT bError THEN 
                (* write successful *)
                bError := FALSE;
                nErrId := 0;
        ELSE 
                (* write failed *)
                bError := fbSdoWriteDInt.bError;
                nErrId := fbSdoWriteDInt.nErrId;
        END_IF

        fbSdoWriteDInt(bExecute := FALSE);
END_IF
/////////////////////////////////////////////////////////
fbSdoWriteBool(
        sNetId          := sNetId,
        nSlaveAddr      := nSlaveAddr,
        nIndex          := nIndex,
        nSubIndex       := nSubIndex,
        pSrcBuf         := ADR(nValueBool),
        cbBufLen        := SIZEOF(nValueBool),
        bExecute        := bExecute
);

IF NOT fbSdoWriteBool.bBusy THEN
        bExecute := FALSE;
        IF NOT bError THEN 
                (* write successful *)
                bError := FALSE;
                nErrId := 0;
        ELSE 
                (* write failed *)
                bError := fbSdoWriteBool.bError;
                nErrId := fbSdoWriteBool.nErrId;
        END_IF

        fbSdoWriteBool(bExecute := FALSE);
END_IF
/////////////////////////////////////////////////////////

END_FUNCTION_BLOCK

// ---- POUs/FB_ROMTest.TcPOU
FUNCTION_BLOCK FB_ROMTest
VAR_INPUT
END_VAR
VAR_OUTPUT
	ROM_act 			: REAL := 0; (*mm*)
	ROM_mirr 			: REAL := 0; (*mm*)
	ROM_ActMid 			: ULINT := 0; (*cts*)
	ROM_MirrMid 		: ULINT := 0; (*cts*)
END_VAR
VAR
	Flip 				: INT := 1;
	ActPosLim 			: ULINT;
	ActNegLim 			: ULINT;
	MirPosLim 			: ULINT;
	MirNegLim 			: ULINT;
	MtrPosP 			: DINT;
	MtrPosN 			: DINT;
	bLimCap 			: BOOL := FALSE;
END_VAR

(*

1092180 = 500 RPM
2184533 = 1000 RPM

*)

IF GVL_TS.bEnableState = TRUE THEN

(*calculate ROM*)
ROM_act := ULINT_TO_REAL(ActPosLim - ActNegLim)*5E-6;
ROM_mirr := ULINT_TO_REAL(MirPosLim - MirNegLim)*5E-6;
ROM_ActMid := (((ActPosLim - ActNegLim) / 2) + ActNegLim);
ROM_MirrMid := (((MirPosLim - MirNegLim) / 2) + MirNegLim);

IF GVL_TS.bEnableState THEN (*if motor is enabled, start test*)
	
	// If neither limit switch is enabled, move until one is reached
	IF NOT GVL_TS.bLim_pos AND NOT GVL_TS.bLim_neg THEN
		GVL_TS.target_vel := flip*LREAL_TO_DINT((1092180) * 10); // 500 RPM
		//GVL_TS.target_vel := flip*LREAL_TO_DINT((1092180) * 2); // 100 RPM
		bLimCap := FALSE; 
	END_IF
	
	// If positive limit reached, reverse direction and continue
//	IF (GVL_TS.bLim_pos := TRUE) THEN
	IF (GVL_TS.bLim_pos = TRUE) AND (bLimCap = FALSE) THEN
		ActPosLim := GVL_TS.ActEncCount;
		MirPosLim := GVL_TS.MirEncCount;
		MtrPosP := GVL_TS.mtr_pos;
		GVL_TS.target_vel := LREAL_TO_DINT(-(1092180) * 10);
		//GVL_TS.target_vel := LREAL_TO_DINT(-(1092180) * 2);
		Flip := -1;
		bLimCap := TRUE;	
	END_IF
	
	// If negative limit reached, reverse direction and continue
//	IF (GVL_TS.bLim_neg := TRUE) THEN
	IF (GVL_TS.bLim_neg = TRUE) AND (bLimCap = FALSE) THEN
		ActNegLim := GVL_TS.ActEncCount;
		MirNegLim := GVL_TS.MirEncCount;
		MtrPosN := GVL_TS.mtr_pos;
		GVL_TS.target_vel := LREAL_TO_DINT((1092180) * 10);
		//GVL_TS.target_vel := LREAL_TO_DINT((1092180) * 2);
		Flip := 1;
		bLimCap := TRUE;
	END_IF	
END_IF

END_IF

END_FUNCTION_BLOCK

// ---- POUs/FB_SineSweep.TcPOU
FUNCTION_BLOCK FB_SineSweep
VAR_INPUT
END_VAR
VAR_OUTPUT
END_VAR
VAR (*file read/write*)
	fbReadSig				: FB_ReadSig;
	fbSaveData				: FB_SaveData;
	bSaveData				: BOOL; 
	VelCmd					: DINT := 0;
	State					: UDINT;
	k						: UDINT :=1;
	Counter					: UDINT;
	PosCmdArray				: ARRAY[1..60000,1..3] OF UDINT ;
END_VAR

VAR (*Drive variables*)
	pos_rb AT %I*			: DINT;
	vel_rb AT %I*			: DINT;
	vel_target AT %Q*		: DINT;
END_VAR

IF GVL_TS.bEnableState = TRUE THEN

// NetID can be found under "Devices/Device 1 (EtherCAT) -> EtherCAT Tab
fbReadSig(
	sSrcNetId := '10.10.160.129.1.1',  
	sSrcPathName := 'C:\HPTTestStand\HPsinesweep\excitation500Hz_multisine_of500.bin', // .BIN file *MUST* be present in this location!
	bExecute := TRUE, 
	tTimeOut := T#5S,
	Step => State,
	cmd => VelCmd );
	IF (State = 5 AND k <= 60000) THEN
		GVL_TS.target_vel := VelCmd;
		PosCmdArray[k,1] := vel_target;
		PosCmdArray[k,2] := vel_rb;	
		PosCmdArray[k,3] := pos_rb;
		k := k+1;
	END_IF

IF bSaveData THEN
	fbSaveData(
	sDestNetId := '10.10.160.129.2.1', 
	sDestPathName := 'C:\HPTTestStand\HPsinesweep\test_veloffset5000.bin', // .BIN file *MUST* be present in this location!
	bExecute := TRUE, 
	tTimeOut := T#5S,
	///buffRead := ADR(PosCmdArray),
	cbWriteLen := SIZEOF(PosCmdArray),
	);
END_IF

Counter := Counter + 1;

END_IF

END_FUNCTION_BLOCK

// ---- POUs/FB_ReadSig.TcPOU
FUNCTION_BLOCK FB_ReadSig
VAR_INPUT
	sSrcNetId			: T_AmsNetId;	(* TwinCAT network address of the source file *)
	sSrcPathName		: T_MaxString;	(* Source file path and name *)
	bExecute			: BOOL;			(* Rising edge start fb execution *)
	tTimeOut			: TIME := DEFAULT_ADS_TIMEOUT;(* Max. ADS timeout time *)
END_VAR
VAR_OUTPUT
	bBusy				:BOOL;(* TRUE => File copy execution in progress, FALSE => File copy execution idle *)
	bError				:BOOL;(* TRUE => Error, FALSE => No error *)
	Step				:UDINT := 0;(* State *)
	nErrId				:UDINT :=0; (*Err ID*)
	cmd					: DINT := 0;
END_VAR
VAR
	fbFileOpen			:FB_FileOpen;
	fbFileClose			:FB_FileClose;
	fbFileRead			: FB_FileRead;
	RisingEdge			: R_TRIG;
	hSrcFile			: UINT	:= 0;(* File handle of the source file *)
//	Step				: DWORD;
	cbReadLength		: UDINT := 0;
	counter				: UDINT := 0;
	k					: UDINT := 0;
	buffRead			: ARRAY[1..60000] OF DINT ;(* Buffr *)
END_VAR

bExecute := MAIN.tglSine;

IF k < 60000 THEN

RisingEdge(CLK:=bExecute);

IF fbFileRead.bEOF THEN
	Step := 50;
END_IF

CASE Step OF
	0:	(* Idle state *)
		IF RisingEdge.Q THEN
			bBusy := TRUE;
			bError:= FALSE;
			nErrId:=0;
			Step := 1;
			cbReadLength:=0;
			hSrcFile:=0;
		END_IF

	1:	(* Open source file *)
		fbFileOpen( bExecute := TRUE );
		fbFileOpen( sNetId := sSrcNetId, sPathName := sSrcPathName,
					nMode := FOPEN_MODEREAD,
					ePath := PATH_GENERIC, tTimeout := tTimeOut, bExecute := TRUE );
//		Step := Step + 1;
(*
	2:
		fbFileOpen( bExecute := TRUE );
		IF NOT fbFileOpen.bBusy THEN
			IF fbFileOpen.bError THEN
				nErrId := fbFileOpen.nErrId;
				bError := TRUE;
				Step := 50;
			ELSE
				hSrcFile := fbFileOpen.hFile;
				Step := Step + 1;
			END_IF
		END_IF
	3:	(* Read data from source file *)
		cbReadLength := 0;
		fbFileRead( bExecute:= TRUE );
		fbFileRead( sNetId:=sSrcNetId, hFile:=hSrcFile,
					pReadBuff:= ADR(buffRead), cbReadLen:= SIZEOF(buffRead),
					bExecute:=TRUE, tTimeout:=tTimeOut );
		Step := Step + 1;
	4:
		fbFileRead( bExecute:= TRUE );
		IF NOT fbFileRead.bBusy THEN
			IF fbFileRead.bEOF THEN (* Check if the EOF flag is set *)
					Step := 50;	(* Cleanup: close the destination and source files *)
			ELSE
				counter := counter+1;
				cbReadLength := fbFileRead.cbRead;
				Step := 3;
			END_IF
			IF fbFileRead.bError THEN
				nErrId := fbFileRead.nErrId;
				bError := TRUE;
				Step := 50;

			END_IF
		END_IF

	40: (* Close source file *)
		fbFileClose( bExecute := TRUE );
		fbFileClose( sNetId:=sSrcNetId, hFile:=hSrcFile, bExecute:=TRUE, tTimeout:=tTimeOut );
		Step := Step + 1;
	41:
		fbFileClose( bExecute := TRUE );
		IF NOT fbFileClose.bBusy THEN
			IF fbFileClose.bError THEN
				nErrId := fbFileClose.nErrId;
				bError := TRUE;
			END_IF
			Step := 50;
			hSrcFile := 0;
		END_IF
	
	// send the command	
	5: 
		k := k+1;
		IF k <= 60000 THEN
			cmd := buffRead[k];
			step := 5;
		ELSE
			step := 0;
		END_IF
		
	50: (* Error or ready => Cleanup *)
		IF (hSrcFile <> 0 ) THEN
			Step := 40; (* Close the source file *)
		ELSE
			Step := 5;	(* Ready *)
			bBusy := FALSE;
		END_IF
*)
END_CASE

ELSE

	//MAIN.tglSine := FALSE;

END_IF

END_FUNCTION_BLOCK

// ---- POUs/FB_SaveData.TcPOU
FUNCTION_BLOCK FB_SaveData
VAR_INPUT
	//sSrcNetId			: T_AmsNetId;	(* TwinCAT network address of the source file *)
	sDestNetId			: T_AmsNetId;	(* TwinCAT network address of the destination file *)
	sDestPathName		: T_MaxString;  (* Destination file path and name *)
	bExecute			: BOOL;			(* Rising edge start fb execution *)
	tTimeOut			: TIME := DEFAULT_ADS_TIMEOUT;(* Max. ADS timeout time *)
	buffRead			: PVOID;
	cbWriteLen			: UDINT;
END_VAR
VAR_OUTPUT
	bBusy				:BOOL;(* TRUE => File copy execution in progress, FALSE => File copy execution idle *)
	bError				:BOOL;(* TRUE => Error, FALSE => No error *)
	nErrId				:UDINT;(* Error code *)
END_VAR
VAR
	fbFileOpen			:FB_FileOpen;
	fbFileClose			:FB_FileClose;
	fbFileWrite			: FB_FileWrite;
	RisingEdge			: R_TRIG;
	hDestFile			: UINT	:= 0;(* File handle of the source file *)
	Step				: DWORD;
	cbReadLength		: UDINT := 0;
	//k					: UDINT := 0;
END_VAR

RisingEdge(CLK:=bExecute);

CASE Step OF
	0:	(* Idle state *)
		IF RisingEdge.Q THEN
			bBusy := TRUE;
			bError:= FALSE;
			nErrId:=0;
			Step := 1;
			cbReadLength:=0;
			hDestFile:=0;
		END_IF


	1:	(* Open destination file *)
		fbFileOpen( bExecute := FALSE );
		fbFileOpen( sNetId := sDestNetId, sPathName := sDestPathName,
					nMode := FOPEN_MODEWRITE OR FOPEN_MODEBINARY,
					ePath := PATH_GENERIC, tTimeout := tTimeOut, bExecute := TRUE );
		Step := Step+1;
	2:
		fbFileOpen( bExecute := FALSE );
		IF NOT fbFileOpen.bBusy THEN
			IF fbFileOpen.bError THEN
				nErrId := fbFileOpen.nErrId;
				bError := TRUE;
				Step := 50;
			ELSE
				hDestFile := fbFileOpen.hFile;
				Step := Step + 1;
			END_IF
		END_IF



	3:	(* Write data to destination file *)
		fbFileWrite( bExecute := FALSE );
		fbFileWrite( sNetId:=sDestNetId, hFile:=hDestFile,
					pWriteBuff:= buffRead, cbWriteLen:= cbWriteLen,
					bExecute:=TRUE, tTimeout:=tTimeOut );
		Step := Step + 1;
	4:
		fbFileWrite( bExecute := FALSE );
		IF NOT fbFileWrite.bBusy THEN
			IF fbFileWrite.bError THEN
				nErrId := fbFileWrite.nErrId;
				bError := TRUE;
				Step := 50;
			ELSE
				Step := 50;
			END_IF
		END_IF

	30:	(* Close the destination file *)
		fbFileClose( bExecute := FALSE );
		fbFileClose( sNetId:=sDestNetId, hFile:=hDestFile, bExecute:=TRUE, tTimeout:=tTimeOut );
		Step := Step + 1;
	31:
		fbFileClose( bExecute := FALSE );
		IF NOT fbFileClose.bBusy THEN
			IF fbFileClose.bError THEN
				nErrId := fbFileClose.nErrId;
				bError := TRUE;
			END_IF
			Step := 50;
			hDestFile := 0;
		END_IF



	50: (* Error or ready => Cleanup *)
		IF ( hDestFile <> 0 ) THEN
			Step := 30; (* Close the destination file*)
		ELSE
			Step := 0;	(* Ready *)
			bBusy := FALSE;
		END_IF

END_CASE

END_FUNCTION_BLOCK

// ---- POUs/FB_TriForce.TcPOU
FUNCTION_BLOCK FB_TriForce
VAR_INPUT
	Slope 					: DINT; 
	Force					: UINT;
	Cycles					: INT;
	Counter					: DINT;
	Channel1Command			: REAL := 0;
	Channel2Command			: REAL := 0;
END_VAR
VAR_OUTPUT
	CyclesOut				: INT := 0;
END_VAR
VAR

END_VAR







(*

__________________________††¥¥
_________________________††††¥¥
________________________††††††¥¥
_______________________††††††††¥¥
______________________††††††††††¥¥
_____________________††††††††††††¥¥
____________________††††††††††††††¥¥
___________________††††††††††††††††¥¥
__________________††††††††††††††††††¥¥
_________________††††††††††††††††††††¥¥
________________††††††††††††††††††††††¥¥
_______________††††††††††††††††††††††††¥¥
______________††††††††††††††††††††††††††¥¥
_____________††††††††††††††††††††††††††††¥¥
____________††¥¥¥¥¥¥¥¥¥¥¥¥¥¥¥¥¥¥¥¥¥¥¥¥¥¥††¥¥
___________††††¥¥¯¯¯¯¯¯¯¯¯¯¯¯¯¯¯¯¯¯¯¯¯¯††††¥¥
__________††††††¥¥¯¯¯¯¯¯¯¯¯¯¯¯¯¯¯¯¯¯¯¯††††††¥¥
_________††††††††¥¥¯¯¯¯¯¯¯¯¯¯¯¯¯¯¯¯¯¯††††††††¥¥
________††††††††††¥¥¯¯¯¯¯¯¯¯¯¯¯¯¯¯¯¯††††††††††¥¥
_______††††††††††††¥¥¯¯¯¯¯¯¯¯¯¯¯¯¯¯††††††††††††¥¥
______††††††††††††††¥¥¯¯¯¯¯¯¯¯¯¯¯¯††††††††††††††¥¥
_____††††††††††††††††¥¥¯¯¯¯¯¯¯¯¯¯††††††††††††††††¥¥
____††††††††††††††††††¥¥¯¯¯¯¯¯¯¯††††††††††††††††††¥¥
___††††††††††††††††††††¥¥¯¯¯¯¯¯††††††††††††††††††††¥¥
__††††††††††††††††††††††¥¥¯¯¯¯††††††††††††††††††††††¥¥
_††††††††††††††††††††††††¥¥¯¯††††††††††††††††††††††††¥¥
††††††††††††††††††††††††††††††††††††††††††††††††††††††¥¥
¯¥¥¥¥¥¥¥¥¥¥¥¥¥¥¥¥¥¥¥¥¥¥¥¥¥¥¥¥¥¥¥¥¥¥¥¥¥¥¥¥¥¥¥¥¥¥¥¥¥¥¥¥¥¥¥¥
____________¶¶3333¶___¶¶¶¶ÿÿÿÿ¶¶¶¶___¶3333¶¶
____________¶¶33333¶_¶ÿÿÿÿÿÿÿÿÿÿÿÿ¶_¶33333¶¶
____________¶¶¶¶¶¶¶¶ÿÿ¶¶¶¶¶¶¶¶¶¶¶¶ÿÿ¶¶¶¶¶¶¶¶
____________¶¶0000¶¶¶77777777777777¶¶¶0000¶¶
____________¶¶0000¶¶7¶¶¶¶¶¶¶¶¶¶¶¶¶¶7¶¶0000¶¶
_____________¶¶000¶¶¶a¯¯¶¶aaaa¶¶¯¯a¶¶¶000¶¶
_____________¶¶000¶¶aa¯¯¶¶aaaa¶¶¯¯aa¶¶000¶¶
______________¶¶00¶¶aaa¯¯aaaaaa¯¯aaa¶¶00¶¶
_______________¶¶000¶¶aaaaaaaaaaaa¶¶000¶¶
________________¶¶00¶¶¶¶aaaaaaaa¶¶¶¶00¶¶
_________________¶¶88888¶¶¶¶¶¶¶¶88888¶¶
__________________¶¶8855888888885588¶¶
__________________¶¶8855555555555588¶¶
________________¶¶11¶¶888855558888¶¶11¶¶
______________¶¶88881111¶¶1111¶¶11118888¶¶
______________¶¶¶¶¶¶8888111111118888¶¶¶¶¶¶
____________¶¶ƒƒ§§¶¶¶¶¶¶88888888¶¶¶¶¶¶§§ƒƒ¶¶
____________¶¶ƒƒƒƒ§§¶¶¯¶¶¶¶¶¶¶¶¶¶¯¶¶§§ƒƒƒƒ¶¶

____________¶¶¶¶¶¶¶¶¶______________¶¶¶¶¶¶¶¶¶


*)

(*
Routine to apply a triangle wave shaped force via the pneumatic piston on the test stand
to the hardpoint

12/15/20 - CHANGED THE FORCE APPLIED TO A SAWTOOTH WAVE; CODE WAS LEFT IN FOR A TRIANGLE WAVE IN CASE A ROLLBACK IS DESIRED

03/03/21 - CHANGED THE FORCE TO ONLY BE APPLIED TO CHANNEL 2, CHANNEL ONE VALUE SET TO CAUSE FORCE VALUE TO PASS THRU ZERO

03/05/21 - ADDED CODE FOR OPTION TO PERFORM BOTH STIFFNESS AND BREAKAWAY TESTS DEPENDING ON WHAT IS (UN)COMMENTED OUT; REMOVED SAWTOOTH WAVE CODE\\

03/29/21 - ADDED CODE TO APPLY FORCE  BETWEEN APPROXIMATELY +/- 300N IN ORDER TO OBSERVE BEHAVIOR OF SMALL DISPLACEMENTS ON HARDPOINTS

08/11/21 - REMOVED REDUNDENT CODE, MADE PARTIONS EASIER TO LOCATE FOR (UN)COMMENTING CODE FOR CHANGING TESTS

10/07/21 - REMOVED "SUPER SOAKER" EFFECT TEST, REORGANIZED TEST ORDER FOR EASE OF CHANGING TESTS

2/27/22 - Condensed everything down to single function block for both breakaway and stiffness
*)

(*=====================================================================================================================================================*)

// For the first quarter of the routine, apply a force one direction fully using one air valve
IF Counter <= 4*Slope THEN
	IF Counter < Slope THEN
		GVL_TS.AirOut2 := REAL_TO_INT(Channel2Command/10*Force); // The dividand multiplle is what controls the force; 7500 => 750N;
		Channel2Command := Channel2Command + 10/DINT_TO_REAL(Slope);
		GVL_TS.AirOut1 := 0;

// For the second quarter of the routine, back the force back off until we are at our starting point
	ELSIF (Counter >= Slope AND Counter < 2*Slope)  THEN
		GVL_TS.AirOut2 := REAL_TO_INT(Channel2Command/10*Force);
		Channel2Command := Channel2Command - 10/DINT_TO_REAL(Slope);
		GVL_TS.AirOut1 := 0;

// For the third quarter of the routine, apply the force in the opposite direction using the other air valve
	ELSIF (Counter >= 2*Slope AND Counter < 3*Slope) THEN
		GVL_TS.AirOut1 := REAL_TO_INT(Channel1Command/10*Force);
		Channel1Command := Channel1Command + 10/DINT_TO_REAL(Slope);
		GVL_TS.AirOut2 := 0;

// For the final quarter of the routine, back the force back off until we are again at our starting point
	ELSIF Counter >= 3*Slope THEN
		GVL_TS.AirOut1 := REAL_TO_INT(Channel1Command/10*Force);
		Channel1Command := Channel1Command - 10/DINT_TO_REAL(Slope);
		GVL_TS.AirOut2 := 0;
	END_IF
		
	// Increment the Counter used to step through the routine
	Counter := Counter +1;
	
	// If the Counter is greater than the number of steps we wish to use to run the test, reset to 0
	IF Counter > 4*Slope THEN
		Counter := 0;
		Cycles := Cycles + 1;
	END_IF

	CyclesOut := Cycles;
END_IF

END_FUNCTION_BLOCK

// ---- POUs/FB_PLoop.TcPOU
FUNCTION_BLOCK FB_PLoop
VAR_INPUT
	fSetpointValue					: REAL ;
END_VAR
VAR_OUTPUT
END_VAR
VAR
	fbPID 							: FB_CTRL_PID;
	stCTRL_PID_PARAMS				: ST_CTRL_PID_PARAMS;
	eErrorId						: E_CTRL_ERRORCODES;
	eMode							: E_CTRL_MODE;
	//fActualValue					: REAL;
	fManSyncValue					: REAL;
	fOut							: REAL;
	//pos_offset					: REAL ;
	//pos_cmd						: REAL ;
	//mir_adjusted					: REAL;
	bHold							: BOOL;
	bError							: BOOL;
	bARWactive						: BOOL;
	bSync							: BOOL;
	bInit							: BOOL	:= TRUE;
END_VAR

IF bInit THEN
	(* init parameter struct *)
	stCTRL_PID_PARAMS.tCtrlCycleTime		:= T#10ms;
	stCTRL_PID_PARAMS.tTaskCycleTime		:= T#10ms;
	stCTRL_PID_PARAMS.fKp					:= 5000.0;			(* proportional gain Kp				*)
	stCTRL_PID_PARAMS.tTn					:= T#0MS;		(*  Tn								*)
	stCTRL_PID_PARAMS.tTv					:= T#0MS;			(*  Tv								*)
	stCTRL_PID_PARAMS.tTd					:= T#0MS;			(*  Td								*)
	stCTRL_PID_PARAMS.fOutMaxLimit			:= (10921800);	(* maximum output limit				*)
	stCTRL_PID_PARAMS.fOutMinLimit			:= (-10921800);	(* minimum output limit				*)
	stCTRL_PID_PARAMS.bDInTheFeedbackPath	:= FALSE;
	stCTRL_PID_PARAMS.bDInTheFeedbackPath	:= FALSE;
	stCTRL_PID_PARAMS.bARWOnIPartOnly		:= TRUE;

	(* set the mode to ACTIVE --> normal operation *)
	eMode := eCTRL_MODE_ACTIVE;

	(* reset the init flag *)
	bInit := FALSE;
END_IF

GVL_TS.control_word := 31;

(* call controller *)
fbPID(			fSetpointValue		:= fSetpointValue ,
				fActualValue		:= GVL_TS.ActEncCount,
				fManSyncValue		:= fManSyncValue,
				bSync				:= bSync,
				eMode				:= eMode,
				bHold				:= bHold,
				stParams			:= stCTRL_PID_PARAMS,
				fOut				=> fOut,
				bARWactive			=> bARWactive,
				eErrorId			=> eErrorId,
				bError				=> bError
				);
				
GVL_TS.target_vel := TO_DINT(fbPID.fOut);
GVL_TS.Pdiff := GVL_TS.ActEncCount - fSetpointValue;

END_FUNCTION_BLOCK

// ---- POUs/FB_BinToVer.TcPOU
FUNCTION_BLOCK FB_BinToVer
VAR_INPUT
	BinInput 			: UINT;
END_VAR
VAR_OUTPUT
	MtrErrArr 			: ARRAY[0..15] OF BOOL;
END_VAR
VAR
END_VAR

// Read in status word from drive amp, read it out bit-wise, write each bit to a corresponding array position, and pass
// the entire array back for the main program to be able to read out and set the verbose error messages on the HMI

MtrErrArr[0] := BinInput.0;
MtrErrArr[1] := BinInput.1;
MtrErrArr[2] := BinInput.2;
MtrErrArr[3] := BinInput.3;
MtrErrArr[4] := BinInput.4;
MtrErrArr[5] := BinInput.5;
MtrErrArr[6] := BinInput.6;
MtrErrArr[7] := BinInput.7;
MtrErrArr[8] := BinInput.8;
MtrErrArr[9] := BinInput.9;
MtrErrArr[10] := BinInput.10;
MtrErrArr[11] := BinInput.11;
MtrErrArr[12] := BinInput.12;
MtrErrArr[13] := BinInput.13;
MtrErrArr[14] := BinInput.14;
MtrErrArr[15] := BinInput.15;

END_FUNCTION_BLOCK

// ---- POUs/FB_SerialCom.TcPOU
FUNCTION_BLOCK FB_SerialCom
VAR_IN_OUT
	TxBuffer			: ComBuffer;
	RxBuffer			: ComBuffer;
END_VAR
VAR
	fbReceive			: ReceiveString;
	sReceivedString		: STRING;
	bStringReceived		: BOOL;
	bReceiveBusy		: BOOL;
	bReceiveError		: BOOL;
	eReceiveErrorID		: ComError_t;
	bReceiveTimeout		: BOOL;
END_VAR
VAR_OUTPUT
	sHeidOut 			: STRING;
	Error				: BOOL := FALSE;
END_VAR

//	Receive string data:
//	The block receives any data strings beginning with a STX ($02) and ending with an ETX ($03) character.	
fbReceive(
	Prefix:= '',
	Suffix:= '',
	Timeout:= T#1s,
	ReceivedString := sHeidOut,
	RXbuffer:= RxBuffer,
	StringReceived=> bStringReceived,
	Busy => bReceiveBusy,
	Error => ,
	RxTimeout => bReceiveTimeout );
IF fbReceive.Error <> COMERROR_NOERROR THEN
	eReceiveErrorID := fbReceive.Error;
	//Error := TRUE;
END_IF

END_FUNCTION_BLOCK

// ---- POUs/FB_HeidConv.TcPOU
FUNCTION_BLOCK FB_HeidConv
VAR_INPUT
	sHeidIn 			: STRING;
END_VAR
VAR_OUTPUT
	s1 					: STRING;
	s2 					: STRING;
	s3 					: STRING;
	s4 					: STRING;
END_VAR
VAR
	PosA 				: INT;
	PosB 				: INT;
	PosC 				: INT;
	PosD 				: INT;
	PosE 				: INT;
END_VAR

// Strip out "A" measurement"
PosA := FIND(sHeidIn, 'A');
PosB := FIND(sHeidIn, 'B');
s1 := sHeidIn;
s1 := DELETE(sHeidIn, LEN(sHeidIn) - PosB + 1, posB);
s1 := DELETE(s1, PosA, 1);


// Strip out "B" measurement
PosB := FIND(sHeidIn, 'B');
PosC := FIND(sHeidIn, 'C');
s2 := sHeidIn;
s2 := DELETE(sHeidIn, LEN(sHeidIn) - PosC + 1, PosC);
s2 := DELETE(s2, PosB, 1);

// Strip out "C" measurement"
PosC := FIND(sHeidIn, 'C');
PosD := FIND(sHeidIn, 'D');
s3 := sHeidIn;
s3 := DELETE(sHeidIn, LEN(sHeidIn) - PosD + 1, PosD);
s3 := DELETE(s3, PosC, 1);

// Strip out "D" measurement"
PosD := FIND(sHeidIn, 'D');
PosE := FIND(sHeidIn, 'E');
s4 := sHeidIn;
s4 := DELETE(sHeidIn, LEN(sHeidIn) - PosE + 1, PosE);
s4 := DELETE(s4, PosD, 1);

END_FUNCTION_BLOCK

// ---- POUs/FB_PyListener.TcPOU
FUNCTION_BLOCK FB_PyListener
VAR_INPUT
	bExecute			: BOOL := FALSE;
	Initialized 		: BOOL := FALSE;
	Init_State  		: UINT := 0;
END_VAR
VAR_OUTPUT
	bIsBusy				: BOOL;
    ERR             	: BOOL;
    ERRID           	: UDINT;
END_VAR
VAR
	Process         	: NT_StartProcess;
	RisingEdge			: R_TRIG;
	bError          	: BOOL;
    sTargetFilePath     : STRING(255);
    sTargetDirectory    : STRING(255);
    sCommand        	: STRING(255);
    iErrorId            : UDINT; 	
END_VAR

IF NOT Initialized THEN
  (* Initialization State Machine *)
  CASE Init_State OF
    0: (* First step in initialization *)
	
		// File Locations
		sTargetDirectory := 'C:\HPTTestStand_Stiff\attocubes4austin\';
 
		// Build Command String                 
		// Special command indicating command string input
		sCommand := CONCAT(sTargetDirectory, 'AttoCube_LC_Readout.py');      // Execute Python data collection script
        Init_State := Init_State + 1;
	   
    1: (* Second step in initialization *)
		Process(
    	NETID := '',                    					// Local System
		//PATHSTR := 'C:\ProgramData\Anaconda3\python.exe',   // Path to local cmd executable
		PATHSTR := 'python',
    	COMNDLINE := sCommand,          					// Comnmand to be executed
    	ERR => bError,                   					// Error Output
    	ERRID => iErrorId,                					// Error Id Output
		BUSY => bIsBusy,									// Process is already busy, used to not call multiple instances
		START := TRUE
		);
        Init_State := Init_State + 1;

    2: (* Last step in initialization *)
		Process(START := FALSE);
		bExecute := FALSE;
		RisingEdge.CLK := FALSE;
        Initialized := TRUE;
  END_CASE
END_IF

END_FUNCTION_BLOCK

// ---- POUs/FB_PyListenerStiffness.TcPOU
FUNCTION_BLOCK FB_PyListenerStiffness
VAR_INPUT
	bExecute			: BOOL := FALSE;
	Initialized 		: BOOL := FALSE;
	Init_State  		: UINT := 0;
END_VAR
VAR_OUTPUT
	bIsBusy				: BOOL;
    ERR             	: BOOL;
    ERRID           	: UDINT;
END_VAR
VAR
	Process         	: NT_StartProcess;
	RisingEdge			: R_TRIG;
	bError          	: BOOL;
    sTargetFilePath     : STRING(255);
    sTargetDirectory    : STRING(255);
    sCommand        	: STRING(255);
    iErrorId            : UDINT; 	
END_VAR

IF NOT Initialized THEN
  (* Initialization State Machine *)
  CASE Init_State OF
    0: (* First step in initialization *)
	
		// File Locations
		sTargetDirectory := 'C:\HPTTestStand_Stiff\attocubes4austin\';
 
		// Build Command String                 
		// Special command indicating command string input
		sCommand := CONCAT(sTargetDirectory, 'AttoCube_LC_Readout_Stiff.py');      // Execute Python data collection script
        Init_State := Init_State + 1;
	   
    1: (* Second step in initialization *)
		Process(
    	NETID := '',                    					// Local System
		PATHSTR := 'python',   // Path to local cmd executable
    	COMNDLINE := sCommand,          					// Comnmand to be executed
    	ERR => bError,                   					// Error Output
    	ERRID => iErrorId,                					// Error Id Output
		BUSY => bIsBusy,									// Process is already busy, used to not call multiple instances
		START := TRUE
		);
        Init_State := Init_State + 1;

    2: (* Last step in initialization *)
		Process(START := FALSE);
		bExecute := FALSE;
		RisingEdge.CLK := FALSE;
        Initialized := TRUE;
  END_CASE
END_IF

END_FUNCTION_BLOCK

// ---- POUs/FB_PLCTime.TcPOU
FUNCTION_BLOCK FB_PLCTime
VAR_INPUT
END_VAR
VAR_OUTPUT
	sTime				: STRING;
END_VAR
VAR
	fbGetTime			: NT_GetTime;
	TimeStr				: TIMESTRUCT;
END_VAR

fbGetTime(
	START := TRUE,
	NETID := '',
	TIMESTR => TimeStr
	);
fbGetTime(
	START := FALSE,
	NETID := ''
	);
	
sTime := CONCAT(TO_STRING(TimeStr.wHour), ':'); 
IF TimeStr.wMinute < 10 THEN
	sTime := CONCAT(sTime, '0');
	sTime := CONCAT(sTime, TO_STRING(TimeStr.wMinute));
ELSE
	sTime := CONCAT(sTime, TO_STRING(TimeStr.wMinute));	
END_IF 
sTime := CONCAT(sTime, ':');
IF TimeStr.wSecond < 10 THEN
	sTime := CONCAT(sTime, '0');
	sTime := CONCAT(sTime, TO_STRING(TimeStr.wSecond));
ELSE
	sTime := CONCAT(sTime, TO_STRING(TimeStr.wSecond));	
END_IF
sTime := CONCAT(sTime, '.');
sTime := CONCAT(sTime, TO_STRING(TimeStr.wMilliseconds));

END_FUNCTION_BLOCK

// ---- POUs/FB_PyPosRep.TcPOU
FUNCTION_BLOCK FB_PyPosRep
VAR_INPUT
	bExecute			: BOOL := FALSE;
	Initialized 		: BOOL := FALSE;
	Init_State  		: UINT := 0;
END_VAR
VAR_OUTPUT
	bIsBusy				: BOOL;
    ERR             	: BOOL;
    ERRID           	: UDINT;
END_VAR
VAR
	Process         	: NT_StartProcess;
	RisingEdge			: R_TRIG;
	bError          	: BOOL;
    sTargetFilePath     : STRING(255);
    sTargetDirectory    : STRING(255);
    sCommand        	: STRING(255);
    iErrorId            : UDINT; 	
END_VAR

IF NOT Initialized THEN
  (* Initialization State Machine *)
  CASE Init_State OF
    0: (* First step in initialization *)
	
		// File Locations
		sTargetDirectory := 'C:\HPTTestStand_Stiff\attocubes4austin\';
 
		// Build Command String                 
		// Special command indicating command string input
		sCommand := CONCAT(sTargetDirectory, 'AttoCube_PosRep_Readout_3.py');      // Execute Python data collection script
        //sCommand := CONCAT(sTargetDirectory, 'Position_Move_Test.py');
		Init_State := Init_State + 1;
	   
    1: (* Second step in initialization *)
		Process(
    	NETID := '',                    					// Local System
		PATHSTR := 'python',   // Path to local cmd executable
    	COMNDLINE := sCommand,          					// Comnmand to be executed
    	ERR => bError,                   					// Error Output
    	ERRID => iErrorId,                					// Error Id Output
		BUSY => bIsBusy,									// Process is already busy, used to not call multiple instances
		START := TRUE
		);
        Init_State := Init_State + 1;

    2: (* Last step in initialization *)
		Process(START := FALSE);
		bExecute := FALSE;
		RisingEdge.CLK := FALSE;
        Initialized := TRUE;
  END_CASE
END_IF

END_FUNCTION_BLOCK

// ---- POUs/FB_ClearFault.TcPOU
FUNCTION_BLOCK FB_ClearFault
VAR_INPUT
	bExecute : BOOL := FALSE;
	slv_addr : UINT := 0;
END_VAR
VAR_OUTPUT
	state : INT := 0;
	
	bError : BOOL;
	
END_VAR
VAR
	fbSdoWrite : FB_EcCoESdoWrite;
	nErrID : UDINT :=0;
	sdo_address: UINT := 16#8006;
	subIndex: BYTE := 1;
	value : INT := 1;
END_VAR

fbSdoWrite(
        sNetId          := MAIN.sNetId_local,
        //nSlaveAddr      := nSlaveAddr,
		nSlaveAddr :=   slv_addr,
        nIndex          := sdo_address,
        nSubIndex       := subIndex,
        pSrcBuf         := ADR(value),
        cbBufLen        := SIZEOF(value),
        bExecute        := bExecute
);
state := 1;
IF NOT fbSdoWrite.bBusy THEN
        bExecute := FALSE;
		//done	:= TRUE;
        IF NOT fbSdoWrite.bError THEN 
                (* write successful *)
                bError := FALSE;
                nErrId := 0;
        ELSE 
                (* write failed *)
                bError := fbSdoWrite.bError;
                nErrId := fbSdoWrite.nErrId;
        END_IF
        fbSdoWrite(bExecute := FALSE);
		state := 0;
END_IF

END_FUNCTION_BLOCK

// ---- POUs/FB_ReadNcyl.TcPOU
FUNCTION_BLOCK FB_ReadNcyl
VAR_INPUT
	bExecute : BOOL := FALSE;
	slv_addr : UINT := 0;
END_VAR
VAR_OUTPUT
	state : INT := 0;
	bError : BOOL;
	value : UINT;
	
END_VAR
VAR
	fbSdoRead : FB_EcCoESdoRead;
	nErrID : UDINT :=0;
	sdo_address: UINT := 16#8005;
	subIndex: BYTE := 5;
	
END_VAR

fbSdoRead(
        sNetId          := MAIN.sNetId_local,
        //nSlaveAddr      := nSlaveAddr,
		nSlaveAddr :=   slv_addr,
        nIndex          := sdo_address,
        nSubIndex       := subIndex,
        pDstBuf         := ADR(value),
        cbBufLen        := SIZEOF(value),
        bExecute        := bExecute
);
state := 1;
IF NOT fbSdoRead.bBusy THEN
        bExecute := FALSE;
		//done	:= TRUE;
        IF NOT fbSdoRead.bError THEN 
                (* write successful *)
                bError := FALSE;
                nErrId := 0;
        ELSE 
                (* write failed *)
                bError := fbSdoRead.bError;
                nErrId := fbSdoRead.nErrId;
        END_IF
        fbSdoRead(bExecute := FALSE);
		state := 0;
END_IF

END_FUNCTION_BLOCK

// ---- POUs/FB_ReadAlias.TcPOU
FUNCTION_BLOCK FB_ReadAlias
VAR_INPUT
	bExecute : BOOL := FALSE;
	slv_addr : UINT := 0;
END_VAR
VAR_OUTPUT
	state : INT := 0;
	bError : BOOL;
	value : UDINT := 0;
	
END_VAR
VAR
	fbSdoRead : FB_EcCoESdoRead;
	nErrID : UDINT :=0;
	sdo_address: UINT := 16#8008;
	subIndex: BYTE := 1;
	
END_VAR

fbSdoRead(
        sNetId          := MAIN.sNetId_local,
        //nSlaveAddr      := nSlaveAddr,
		nSlaveAddr :=   slv_addr,
        nIndex          := sdo_address,
        nSubIndex       := subIndex,
        pDstBuf         := ADR(value),
        cbBufLen        := SIZEOF(value),
        bExecute        := bExecute
);
state := 1;
IF NOT fbSdoRead.bBusy THEN
        bExecute := FALSE;
		//done	:= TRUE;
        IF NOT fbSdoRead.bError THEN 
                (* write successful *)
                bError := FALSE;
                nErrId := 0;
        ELSE 
                (* write failed *)
                bError := fbSdoRead.bError;
                nErrId := fbSdoRead.nErrId;
        END_IF
        fbSdoRead(bExecute := FALSE);
		state := 0;
END_IF

END_FUNCTION_BLOCK

// ---- POUs/FB_readtextfile.TcPOU
FUNCTION_BLOCK FB_readtextfile
VAR_INPUT
	bRead : BOOL :=FALSE;
	sFileName : T_MaxString ;
END_VAR
VAR_OUTPUT
	step			: DWORD 	:= 0;
	output : ARRAY[1.. GVL_TS.max_rows] OF REAL;
END_VAR
VAR
	//bRead			: BOOL := FALSE;(* Rising edge starts program execution *)
	//sNetId			: T_AmsNetId := '10.10.16.19.1.1';	(* TwinCAT system network address *)
	sNetID			: T_AmsNetId := '10.134.198.192.2.1';
	//sFileName		: T_MaxString ;
	//sFileName		: T_MaxString := 'C:\Users\tranka\Documents\TcXaeShell\signals\sinesweep_f1_50Hz_dt_1000Hz_amp15N_offset0.csv';(* CSV source file path and name *)
	sCSVLine		: T_MaxString := '';(* Single CSV text line (row, record), we are using string as record buffer (your are able to see read fields)  *)
	sCSVField		: T_MaxString := '';(* Single CSV field value (column, record field) *)
	bBusy			: BOOL;
	bError			: BOOL;
	nErrId			: UDINT;
	nRow	 		: UDINT 	:= 1;(* Row number (record) *)
	nColumn			: UDINT 	:= 0;(* Column number (record field) *)
	hFile			: UINT		:= 0;(* File handle of the source file *)
	
	fbFileOpen		: FB_FileOpen;(* Opens file *)
	fbFileClose		: FB_FileClose;(* Closes file *)
	fbFileGets		: FB_FileGets;(* Reads one record (line) *)
	fbReader		: FB_CSVMemBufferReader;(* Helper function block used to parse CSV data bytes (single record line) *)

	database		: ARRAY[1.. GVL_TS.max_rows] OF STRING(100);(* Target PLC database *)
	MAX_CSV_ROWS: UDINT := GVL_TS.max_rows;
	//MAX_CSV_COLUMNS: UDINT:= 1;
END_VAR

CASE step OF
	0:	(* Wait for rising edge at bRead variable *)
		IF bRead THEN
			bRead 	:= FALSE;
			bBusy 	:= TRUE;
			bError	:= FALSE;
			nErrId	:= 0;
			hFile	:= 0;
			nRow	:= 1;
			//nColumn	:= 0;
			MEMSET( ADR( database ), 0, SIZEOF( database ) );
			step 		:= 1;
		END_IF

	1:	(* Open source file *)
		fbFileOpen(  bExecute := FALSE  );
		fbFileOpen( sNetId := sNetId, sPathName := sFileName, nMode := FOPEN_MODEREAD OR FOPEN_MODETEXT,(* Open file in TEXT mode! *)
					ePath := PATH_GENERIC, bExecute := TRUE );
		step := 2;

	2:(* Wait until open not busy *)
		fbFileOpen( bExecute := FALSE, bError => bError, nErrID => nErrID, hFile => hFile );
		IF NOT fbFileOpen.bBusy THEN
			IF NOT fbFileOpen.bError THEN
				step := 3;
			ELSE(* Error: file not found? *)
				step := 100;
			END_IF
		END_IF

	3:	(* Read single line (record) *)
		fbFileGets( bExecute := FALSE );
		fbFileGets( sNetId := sNetId, hFile := hFile, bExecute := TRUE );
		step := 4;

	4:(* Wait until read not busy *)
		fbFileGets( bExecute := FALSE, bError => bError, nErrID => nErrID, sLine => sCSVLine );
		IF NOT fbFileGets.bBusy THEN
			IF NOT fbFileGets.bError THEN
				IF fbFileGets.bEOF THEN
					step := 10;(* End of file reached => Close source file *)
				ELSE

					(* FB_FileGets returns text line without the CR (carriage return) character.
					We have to restore the CR character (replace the $L character with $R$L characters) *)
					IF RIGHT( sCSVLine, 1 ) = '$L' THEN
						sCSVLine := REPLACE( sCSVLine, '$R$L', 2, LEN( sCSVLine ) );
					END_IF

					step := 5;
				END_IF
			ELSE(* Error *)
				step := 100;
			END_IF
		END_IF

	5:(* Parse single line (record) *)
		fbReader.eCmd := eEnumCmd_First;(* Read first field value *)
		REPEAT
			fbReader( pBuffer := ADR( sCSVLine ), cbBuffer := SIZEOF( sCSVLine ), getValue => sCSVField );
			IF fbReader.bOk THEN
				fbReader.eCmd := eEnumCmd_Next;(* Read next field value *)

				IF ( nRow <= MAX_CSV_ROWS ) THEN
					//IF ( nColumn <= MAX_CSV_COLUMNS ) THEN
						database[nRow] := CSVFIELD_TO_STRING( sCSVField, FALSE );(* TODO: Save or use the field value in your application *)
						output[nRow] := STRING_TO_REAL(database[nRow]);
					//END_IF
				END_IF

				//nColumn := nColumn + 1;(* Increment number of read columns *)
				IF fbReader.bCRLF THEN(* CRLF == TRUE => End of reacord reached *)
					nRow 		:= nRow + 1;(* Increment number of read records *)
					//nColumn 	:= 0;(* Reset number of columns *)
				END_IF

			ELSE(* Error: End of record reached or all fields read *)
				step := 3;(* Try to read next line *)
			END_IF
		UNTIL NOT fbReader.bOk
		END_REPEAT

	10:	(* Close source file *)
		fbFileClose( bExecute := FALSE );
		fbFileClose( sNetId := sNetId, hFile := hFile, bExecute := TRUE );
		step := 11;

	11:(* Wait until close not busy *)
		fbFileClose( bExecute := FALSE, bError => bError, nErrID => nErrID );
		IF ( NOT fbFileClose.bBusy ) THEN
			hFile := 0;
			step := 100;
		END_IF

	100: (* Error or ready step => cleanup *)
		IF ( hFile <> 0 ) THEN
			step := 10; (* Close the source file *)
		ELSE
			bBusy := FALSE;
			step := 0;	(* Ready *)
		END_IF

END_CASE

END_FUNCTION_BLOCK

// ---- POUs/FB_WritePWM.TcPOU
FUNCTION_BLOCK FB_WritePWM
VAR_INPUT
	bExecute : BOOL := FALSE;
	slv_addr : UINT := 0;
	value : REAL := 0.0;
END_VAR
VAR_OUTPUT
	state : INT := 0;
	bError : BOOL;
END_VAR
VAR
	fbSdoWrite : FB_EcCoESdoWrite;
	nErrID : UDINT :=0;
	sdo_address: UINT := 16#8001;
	subIndex: BYTE := 7;
END_VAR

fbSdoWrite(
        sNetId          := MAIN.sNetId_local,
        //nSlaveAddr      := nSlaveAddr,
		nSlaveAddr :=   slv_addr,
        nIndex          := sdo_address,
        nSubIndex       := subIndex,
        pSrcBuf         := ADR(value),
        cbBufLen        := SIZEOF(value),
        bExecute        := bExecute
);
state := 1;
IF NOT fbSdoWrite.bBusy THEN
        bExecute := FALSE;
		//done	:= TRUE;
        IF NOT fbSdoWrite.bError THEN 
                (* write successful *)
                bError := FALSE;
                nErrId := 0;
        ELSE 
                (* write failed *)
                bError := fbSdoWrite.bError;
                nErrId := fbSdoWrite.nErrId;
        END_IF
        fbSdoWrite(bExecute := FALSE);
		state := 0;
END_IF

END_FUNCTION_BLOCK

// ---- POUs/FB_CountConv.TcPOU
FUNCTION FB_CountConv : REAL
VAR_INPUT
	COUNTS_IN 			: DINT;
END_VAR
VAR
END_VAR
VAR_OUTPUT
	MEASC_OUT 			: REAL;
	MEASF_OUT 			: REAL;
END_VAR

// Conversion for counts to mm -> distance [resolution (nm) * (nm -> mm) * # of counts]

// Renishaw DIP-SWITCH CONFIG, 12/09/20
// NOTE: CONSULT RENISHAW USER MANUAL FOR SWITCH SETTING CONFIGURATION BREAKDOWN

// Switch Up   Switch Down
//    [0]		  [-]
//    [-]         [o]
//
// 15               1
// [ooo-o---|o--o-o--]
// [---o-ooo|-oo-o-oo]

// Coarse resolution conversion
MEASC_OUT := 79 * 0.000001 * COUNTS_IN;

// Fine resolution conversion
MEASF_OUT := 39.5 * 0.000001 * COUNTS_IN;

END_FUNCTION

// ---- POUs/FB_AirConv.TcPOU
FUNCTION FB_AirConv
VAR_INPUT
	AirIN 				: REAL;
END_VAR
VAR
END_VAR

//Function to convert air control HMI slider values into EL4102 0-10V signal output

// If slider value > 0
IF AirIN > 0 THEN
	GVL_TS.AirOut2 := TRUNC_INT((AirIn / 100) * 32767); // Ch1 Output = Postive % of 16bit output value; drop any decimal points
	GVL_TS.AirOut1 := 0;
END_IF

// If slider < 0
IF (AirIn < 0) THEN
	GVL_TS.AirOut1 := TRUNC_INT((AirIn / -100) * 32767); // Same as above, but sign flipped for Ch2
	GVL_TS.AirOut2 := 0;
END_IF

// If Slider value = 0, set both channels to 0
IF (AirIn = 0) THEN
	GVL_TS.AirOut1 := 0;
	GVL_TS.AirOut2 := 0;
END_IF

END_FUNCTION

// ---- POUs/FB_MtrCtrl.TcPOU
FUNCTION FB_MtrCtrl 		: BOOL
VAR_INPUT	
END_VAR
VAR_OUTPUT
	bBtnEnb 			: BOOL;
END_VAR
VAR
	StickyRead 			: UDINT;
	EncoderFaultRead 	: UDINT;
END_VAR

(* 
	-=CONTROL WORD DESCRIPTION=-
	
	BIT 0: ENABLE AMP WHEN HIGH
	BIT 1: ENABLE VOLTAGE WHEN HIGH
	BIT 2: QUICK STEP DISABLE WHEN CLEAR
	BIT 3: ENABLE AMP WHEN HIGH
	BIT 4: OPERATION MODE SPECIFIC
	BIT 5: OPERATION MODE SPECIFIC
	BIT 6: OPERATION MODE SPECIFIC
	BIT 7: RESET FAULT WHEN LOW TO HIGH DETECTED
	BIT 8: HALT WHEN HIGH
	BITS 9-15: RESERVED FOR FUTURE USE
*)

IF GVL_TS.bEnable = TRUE THEN (*Enable the motor*)
	GVL_TS.control_word := 16#0000; // 0, 0x0000, 0b00000000
	GVL_TS.control_word := 16#0080; // 128, 0x0080, 0b10000000
	GVL_TS.control_word := 16#0006; // 6, 0x0006, 0b00000110
	GVL_TS.control_word := 16#0007; // 7, 0x0007, 0b00000111
	GVL_TS.control_word := 16#001F; // 31, 0x001f, 0b00011111
ELSIF GVL_TS.bEnable = FALSE THEN (*disable the motor*)
	GVL_TS.control_word := 2#00000110; //16#0007; // 6, 0x0006, 0b00000110
	GVL_TS.target_vel := 0; // 0, 0x0000, 0b00000000
END_IF


(*
	-=STATUS WORD DESCRIPTION=-
	
	BIT 0: READY TO SWITCH ON
	BIT 1: SWITCHED ON
	BIT 2: OPERATION ENABLED
	BIT 3: (LATCHED, IF SET) FAULT
	BIT 4: VOLTAGE ENABLED
	BIT 5: QUICK STOP; IF CLEAR, AMP IS PERFORMING A QUICK STOP
	BIT 6: SWITCH ON DISABLED
	BIT 7: WARNING
	BIT 8: LAST TRAJECTORY ABORTED
	BIT 9: REMOTE CONTROL ENABLED THROUGH CANopen
	BIT 10: TARGET REACHED; NOT CLEARED UNTIL NEW TRAJECTORY STARTED
	BIT 11: INTERNAL LIMIT ACTIVE
	BIT 12: OPERATION SPECIFIC; POSITION: SET POINT ACKNOWLADGED, VELOCITY: SPEED = 0
	BIT 13: OPERATION SPECIFIC; POSITION: FOLLOWING ERROR, VELOCITY: MAX SLIPPAGE ERROR
	BIT 14: AMP IS PERFORMING A MOVE
	BIT 15: SET WHEN HOME POSITION CAPTURED
*)

IF GVL_TS.status_word.2 = TRUE THEN(*read bit 2 to check if motor is enabled*)
	GVL_TS.bEnableState := TRUE;
	bBtnEnb := TRUE;
ELSE
	GVL_TS.bEnableState := FALSE;
	bBtnEnb := FALSE;
END_IF

IF GVL_TS.bReset THEN
	GVL_TS.control_word := 0; //0x00000000
	GVL_TS.control_word := 16#8F; //0x008f, 0b10000111
	GVL_TS.control_word := 0;
	GVL_TS.TransitionFromQS := 3;
	GVL_TS.StopAbort := 0;
	GVL_TS.ClearLatched2183 := 16#FFFFFFFF;
	GVL_TS.ClearLatched2183 := 16#00000000;
	GVL_TS.ClearLatched2183.7 := 1;
	GVL_TS.ClearLatched2181 := 16#FFFFFFFF;
	GVL_TS.ClearLatched2181 := 16#00000000;
	StickyRead := GVL_TS.Sticky;
	EncoderFaultRead := GVL_TS.EncoderFault;
	GVL_TS.bEnableState := FALSE;
	GVL_TS.bReset := FALSE;
END_IF

(*check limit switches*)
IF (GVL_TS.DIO_status.0) = FALSE AND (GVL_TS.DIO_status.1) = FALSE THEN  // 0x043f0008, 0b100001111110000000000001000
	GVL_TS.bLim_neg := FALSE;
	GVL_TS.bLim_pos := FALSE;
END_IF

IF (GVL_TS.DIO_status.0) = FALSE AND (GVL_TS.DIO_status.1) = TRUE THEN  // 0x043b000a, 0b100001111110000000000001010
	GVL_TS.bLim_neg := FALSE;
	GVL_TS.bLim_pos := TRUE;
END_IF

IF (GVL_TS.DIO_status.0) = TRUE AND (GVL_TS.DIO_status.1) = FALSE  THEN  // 0x04370009, 0b100001111110000000000001001
	GVL_TS.bLim_neg := TRUE;
	GVL_TS.bLim_pos := FALSE;
END_IF

END_FUNCTION
